(* CODESYS project PartX_Codesys

Project tree, tasks and I/O mapping:
  Device : CODESYS Control Win V3 x64, CODESYS, version 3.5.22.10
    application Application
      libraries: Standard, 3.5.22.0 (System); VisuDialogs, * (System); CAA Net Base Services, * (CAA Technical Workgroup)
      task ENIPScannerIOTask (cyclic, interval t#10ms, priority 0) calls EtherNet_IP_Scanner.IOCycle
      task ENIPScannerServiceTask (cyclic, interval t#20ms, priority 30) calls EtherNet_IP_Scanner.ServiceCycle
      task MainTask (cyclic, interval t#20ms, priority 1) calls F001_SR00_MAIN, F002_SR00_MAIN
      task VISU_TASK (cyclic, interval 100 ms, priority 31) calls VisuElems.Visu_Prg
      F001_ROBOT/
        program F001_SR00_MAIN [?]
        program F001_SR02_RBT_ERRORS [?]
        program F001_SR03_STEPS [?]
        program F001_SR04_RBT_INIT [?]
        program F001_SR05_SET_TRF [?]
        program F001_SR06_RBT_MOTIONS [?]
        program F001_SR07_CAMERA [?]
        program F001_SR08_Explicit [ST]
        program F001_SR08_Explicit_Messaging [ST]
        program F001_SR08_ExplicitMessaging [?]
        function block RobotHandshake [ST]
      F002_PART_X/
        program F002_SR00_MAIN [?]
        program F002_SR01_SOCKET_SERVER [ST]
        program F002_SR02_SOCKET_CLIENT [ST]
        program F002_SR03_PARTX [?]: BOUNCE, CLEAR, IDLE, IDLE_Trigger, Manual_ACT, MOVE_FWD, MOVE_MANUAL, MOVE_REV, SCHED, SCHED_ACT
      F020_HMI_Pages/
        visualisation F020_Camera_Robot
        visualisation F020_PartX_Screen
        visualisation Visualization
      F1000_FBs/
        Meca500/
          function block Delay [ST]
          function block GetErrors [ST]
          function block Gripper [ST]
          function block MoveGripper [ST]
          function block MoveJoints [ST]
          function block MoveJointsRel [ST]
          function block MoveJointsVel [ST]
          function block MoveLin [ST]
          function block MoveLinRelTrf [ST]
          function block MoveLinRelWrf [ST]
          function block MoveLinVelTrf [ST]
          function block MoveLinVelWrf [ST]
          function block MovePose [ST]
          function block SetAutoConf [ST]
          function block SetAutoConfTurn [ST]
          function block SetBlending [ST]
          function block SetCartAcc [ST]
          function block SetCartAngVel [ST]
          function block SetCartLinVel [ST]
          function block SetCheckpoint [ST]
          function block SetConf [ST]
          function block SetConfTurn [ST]
          function block SetGripperForce [ST]
          function block SetGripperRange [ST]
          function block SetGripperVel [ST]
          function block SetJointAcc [ST]
          function block SetJointsVelLimit [ST]
          function block SetJointVel [ST]
          function block SetTorqueLimitCfg [ST]
          function block SetTorqueLimits [ST]
          function block SetTrf [ST]
          function block SetValveState [ST]
          function block SetVelTimeout [ST]
          function block SetWrf [ST]
          function block StartProgram [ST]
          Utiliy/
            function block CalculateWRF [ST]
      F1000_UDTs/
        data type E_SchedState
        data type UDT_Explicit
        UDT_Meca500/
          ENUM/
            data type Meca500_DynamicDataTypeID
            data type Meca500_Errors
            data type Meca500_MotionCommandID
          STRUCT/
            data type Meca500
            Meca500_Inputs/
              data type Meca500_DynamicData
              data type Meca500_Inputs
              data type Meca500_Motion
              data type Meca500_MotionStatus
              data type Meca500_RobotStatus
              data type Meca500_Status
              data type Meca500_TimeStamp
            Meca500_Outputs/
              data type Meca500_BrakeControl
              data type Meca500_MotionCommand
              data type Meca500_MotionControl
              data type Meca500_Outputs
              data type Meca500_RobotControl
        data type UDT_PARTX
        data type UDT_Robot
        data type UDT_StepConfig
        data type UDT_SYS
        data type UDT_VS_Series
      F100_VARs/
        global variables GVL
        text list TL_Directions
      program PLC_PRG [ST]
    Ethernet : Ethernet, CODESYS, version 4.2.0.0
        settings: IPAddress = [192,168,0,247]; SubnetMask = [255,255,255,0]; GatewayAddress = [0,0,0,0]; MACAddress = [16#E8,16#97,16#44,16#1A,16#95,16#04]; NetworkInterfaceName = 'Ethernet'; NetworkInterfaceName = "Ethernet"; SaveCommunicationSettings = FALSE; IPAddress = [192,168,0,2]; SubnetMask = [255,255,255,0]; GatewayAddress = [0,0,0,0]
      EtherNet_IP_Scanner : EtherNet/IP Scanner, CODESYS, order no. 1, version 4.8.0.0
        FANUC_Robot : Generic EtherNet/IP device, CODESYS, version 4.6.0.0
            settings: INITIALIZED = TRUE; IP address of Target = [16#C0,16#A8,16#00,16#01]; Keying.Check Device Type = FALSE; Keying.Check Vendor Code = FALSE; Keying.Check Product Code = FALSE; Keying.Check Major Revision = FALSE; Keying.Check Minor Revision = FALSE; RequiredConfigVersion = 50660864; Number of Connections = 1; Connection Settings.Requested packet interval = 32000 µs; Connection Settings.OT Connection Parameters = 18502; Connection Settings.TO Connection Parameters = 18498; Connection Settings.Connection Flags = 1056; Connection Settings.Connection Path Size = 8; Connection Settings.Large OT Connection Parameters = 1207959622; Connection Settings.Large TO Connection Parameters = 1207959618; Connection Path = [16#20,16#04,16#24,16#64,16#2C,16#97,16#2C,16#65]; Heartbeat Multiplier = 1; Input_Param0.ReadOnly = False; Input_Param0.BitSize = 8; Input_Param0.DataSize = 1; Input_Param1.ReadOnly = False; Input_Param1.BitSize = 8; Input_Param1.DataSize = 1; Input_Param2.ReadOnly = False; Input_Param2.BitSize = 8; Input_Param2.DataSize = 1; Input_Param3.ReadOnly = False; Input_Param3.BitSize = 8; Input_Param3.DataSize = 1; Input_Param4.ReadOnly = False; Input_Param4.BitSize = 8; Input_Param4.DataSize = 1; Input_Param5.ReadOnly = False; Input_Param5.BitSize = 8; Input_Param5.DataSize = 1; Input_Param6.ReadOnly = False; Input_Param6.BitSize = 8; Input_Param6.DataSize = 1; Input_Param7.ReadOnly = False;
              Input_Param7.BitSize = 8; Input_Param7.DataSize = 1; Input_Param8.ReadOnly = False; Input_Param8.BitSize = 8; Input_Param8.DataSize = 1; Input_Param9.ReadOnly = False; Input_Param9.BitSize = 8; Input_Param9.DataSize = 1; Input_Param10.ReadOnly = False; Input_Param10.BitSize = 8; Input_Param10.DataSize = 1; Input_Param11.ReadOnly = False; Input_Param11.BitSize = 8; Input_Param11.DataSize = 1; Input_Param12.ReadOnly = False; Input_Param12.BitSize = 8; Input_Param12.DataSize = 1; Input_Param13.ReadOnly = False; Input_Param13.BitSize = 8; Input_Param13.DataSize = 1; Input_Param14.ReadOnly = False; Input_Param14.BitSize = 8; Input_Param14.DataSize = 1; Input_Param15.ReadOnly = False; Input_Param15.BitSize = 8; Input_Param15.DataSize = 1; Input_Param16.ReadOnly = False; Input_Param16.BitSize = 8; Input_Param16.DataSize = 1; Input_Param17.ReadOnly = False; Input_Param17.BitSize = 8; Input_Param17.DataSize = 1; Input_Param18.ReadOnly = False; Input_Param18.BitSize = 8; Input_Param18.DataSize = 1; Input_Param19.ReadOnly = False; Input_Param19.BitSize = 8; Input_Param19.DataSize = 1; Input_Param20.ReadOnly = False; Input_Param20.BitSize = 8;
              Input_Param20.DataSize = 1; Input_Param21.ReadOnly = False; Input_Param21.BitSize = 8; Input_Param21.DataSize = 1; Input_Param22.ReadOnly = False; Input_Param22.BitSize = 8; Input_Param22.DataSize = 1; Input_Param23.ReadOnly = False; Input_Param23.BitSize = 8; Input_Param23.DataSize = 1; Input_Param24.ReadOnly = False; Input_Param24.BitSize = 8; Input_Param24.DataSize = 1; Input_Param25.ReadOnly = False; Input_Param25.BitSize = 8; Input_Param25.DataSize = 1; Input_Param26.ReadOnly = False; Input_Param26.BitSize = 8; Input_Param26.DataSize = 1; Input_Param27.ReadOnly = False; Input_Param27.BitSize = 8; Input_Param27.DataSize = 1; Input_Param28.ReadOnly = False; Input_Param28.BitSize = 8; Input_Param28.DataSize = 1; Input_Param29.ReadOnly = False; Input_Param29.BitSize = 8; Input_Param29.DataSize = 1; Input_Param30.ReadOnly = False; Input_Param30.BitSize = 8; Input_Param30.DataSize = 1; Input_Param31.ReadOnly = False; Input_Param31.BitSize = 8; Input_Param31.DataSize = 1; Input_Param32.ReadOnly = False; Input_Param32.BitSize = 8; Input_Param32.DataSize = 1; Input_Param33.ReadOnly = False; Input_Param33.BitSize = 8; Input_Param33.DataSize = 1;
              Input_Param34.ReadOnly = False; Input_Param34.BitSize = 8; Input_Param34.DataSize = 1; Input_Param35.ReadOnly = False; Input_Param35.BitSize = 8; Input_Param35.DataSize = 1; Input_Param36.ReadOnly = False; Input_Param36.BitSize = 8; Input_Param36.DataSize = 1; Input_Param37.ReadOnly = False; Input_Param37.BitSize = 8; Input_Param37.DataSize = 1; Input_Param38.ReadOnly = False; Input_Param38.BitSize = 8; Input_Param38.DataSize = 1; Input_Param39.ReadOnly = False; Input_Param39.BitSize = 8; Input_Param39.DataSize = 1; Input_Param40.ReadOnly = False; Input_Param40.BitSize = 8; Input_Param40.DataSize = 1; Input_Param41.ReadOnly = False; Input_Param41.BitSize = 8; Input_Param41.DataSize = 1; Input_Param42.ReadOnly = False; Input_Param42.BitSize = 8; Input_Param42.DataSize = 1; Input_Param43.ReadOnly = False; Input_Param43.BitSize = 8; Input_Param43.DataSize = 1; Input_Param44.ReadOnly = False; Input_Param44.BitSize = 8; Input_Param44.DataSize = 1; Input_Param45.ReadOnly = False; Input_Param45.BitSize = 8; Input_Param45.DataSize = 1; Input_Param46.ReadOnly = False; Input_Param46.BitSize = 8; Input_Param46.DataSize = 1; Input_Param47.ReadOnly = False;
              Input_Param47.BitSize = 8; Input_Param47.DataSize = 1; Input_Param48.ReadOnly = False; Input_Param48.BitSize = 8; Input_Param48.DataSize = 1; Input_Param49.ReadOnly = False; Input_Param49.BitSize = 8; Input_Param49.DataSize = 1; Input_Param50.ReadOnly = False; Input_Param50.BitSize = 8; Input_Param50.DataSize = 1; Input_Param51.ReadOnly = False; Input_Param51.BitSize = 8; Input_Param51.DataSize = 1; Input_Param52.ReadOnly = False; Input_Param52.BitSize = 8; Input_Param52.DataSize = 1; Input_Param53.ReadOnly = False; Input_Param53.BitSize = 8; Input_Param53.DataSize = 1; Input_Param54.ReadOnly = False; Input_Param54.BitSize = 8; Input_Param54.DataSize = 1; Input_Param55.ReadOnly = False; Input_Param55.BitSize = 8; Input_Param55.DataSize = 1; Input_Param56.ReadOnly = False; Input_Param56.BitSize = 8; Input_Param56.DataSize = 1; Input_Param57.ReadOnly = False; Input_Param57.BitSize = 8; Input_Param57.DataSize = 1; Input_Param58.ReadOnly = False; Input_Param58.BitSize = 8; Input_Param58.DataSize = 1; Input_Param59.ReadOnly = False; Input_Param59.BitSize = 8; Input_Param59.DataSize = 1; Input_Param60.ReadOnly = False; Input_Param60.BitSize = 8;
              Input_Param60.DataSize = 1; Input_Param61.ReadOnly = False; Input_Param61.BitSize = 8; Input_Param61.DataSize = 1; Input_Param62.ReadOnly = False; Input_Param62.BitSize = 8; Input_Param62.DataSize = 1; Input_Param63.ReadOnly = False; Input_Param63.BitSize = 8; Input_Param63.DataSize = 1; Output_Param0.ReadOnly = False; Output_Param0.BitSize = 8; Output_Param0.DataSize = 1; Output_Param1.ReadOnly = False; Output_Param1.BitSize = 8; Output_Param1.DataSize = 1; Output_Param2.ReadOnly = False; Output_Param2.BitSize = 8; Output_Param2.DataSize = 1; Output_Param3.ReadOnly = False; Output_Param3.BitSize = 8; Output_Param3.DataSize = 1; Output_Param4.ReadOnly = False; Output_Param4.BitSize = 8; Output_Param4.DataSize = 1; Output_Param5.ReadOnly = False; Output_Param5.BitSize = 8; Output_Param5.DataSize = 1; Output_Param6.ReadOnly = False; Output_Param6.BitSize = 8; Output_Param6.DataSize = 1; Output_Param7.ReadOnly = False; Output_Param7.BitSize = 8; Output_Param7.DataSize = 1; Output_Param8.ReadOnly = False; Output_Param8.BitSize = 8; Output_Param8.DataSize = 1; Output_Param9.ReadOnly = False; Output_Param9.BitSize = 8; Output_Param9.DataSize = 1;
              Output_Param10.ReadOnly = False; Output_Param10.BitSize = 8; Output_Param10.DataSize = 1; Output_Param11.ReadOnly = False; Output_Param11.BitSize = 8; Output_Param11.DataSize = 1; Output_Param12.ReadOnly = False; Output_Param12.BitSize = 8; Output_Param12.DataSize = 1; Output_Param13.ReadOnly = False; Output_Param13.BitSize = 8; Output_Param13.DataSize = 1; Output_Param14.ReadOnly = False; Output_Param14.BitSize = 8; Output_Param14.DataSize = 1; Output_Param15.ReadOnly = False; Output_Param15.BitSize = 8; Output_Param15.DataSize = 1; Output_Param16.ReadOnly = False; Output_Param16.BitSize = 8; Output_Param16.DataSize = 1; Output_Param17.ReadOnly = False; Output_Param17.BitSize = 8; Output_Param17.DataSize = 1; Output_Param18.ReadOnly = False; Output_Param18.BitSize = 8; Output_Param18.DataSize = 1; Output_Param19.ReadOnly = False; Output_Param19.BitSize = 8; Output_Param19.DataSize = 1; Output_Param20.ReadOnly = False; Output_Param20.BitSize = 8; Output_Param20.DataSize = 1; Output_Param21.ReadOnly = False; Output_Param21.BitSize = 8; Output_Param21.DataSize = 1; Output_Param22.ReadOnly = False; Output_Param22.BitSize = 8; Output_Param22.DataSize = 1; Output_Param23.ReadOnly = False;
              Output_Param23.BitSize = 8; Output_Param23.DataSize = 1; Output_Param24.ReadOnly = False; Output_Param24.BitSize = 8; Output_Param24.DataSize = 1; Output_Param25.ReadOnly = False; Output_Param25.BitSize = 8; Output_Param25.DataSize = 1; Output_Param26.ReadOnly = False; Output_Param26.BitSize = 8; Output_Param26.DataSize = 1; Output_Param27.ReadOnly = False; Output_Param27.BitSize = 8; Output_Param27.DataSize = 1; Output_Param28.ReadOnly = False; Output_Param28.BitSize = 8; Output_Param28.DataSize = 1; Output_Param29.ReadOnly = False; Output_Param29.BitSize = 8; Output_Param29.DataSize = 1; Output_Param30.ReadOnly = False; Output_Param30.BitSize = 8; Output_Param30.DataSize = 1; Output_Param31.ReadOnly = False; Output_Param31.BitSize = 8; Output_Param31.DataSize = 1; Output_Param32.ReadOnly = False; Output_Param32.BitSize = 8; Output_Param32.DataSize = 1; Output_Param33.ReadOnly = False; Output_Param33.BitSize = 8; Output_Param33.DataSize = 1; Output_Param34.ReadOnly = False; Output_Param34.BitSize = 8; Output_Param34.DataSize = 1; Output_Param35.ReadOnly = False; Output_Param35.BitSize = 8; Output_Param35.DataSize = 1; Output_Param36.ReadOnly = False; Output_Param36.BitSize = 8;
              Output_Param36.DataSize = 1; Output_Param37.ReadOnly = False; Output_Param37.BitSize = 8; Output_Param37.DataSize = 1; Output_Param38.ReadOnly = False; Output_Param38.BitSize = 8; Output_Param38.DataSize = 1; Output_Param39.ReadOnly = False; Output_Param39.BitSize = 8; Output_Param39.DataSize = 1; Output_Param40.ReadOnly = False; Output_Param40.BitSize = 8; Output_Param40.DataSize = 1; Output_Param41.ReadOnly = False; Output_Param41.BitSize = 8; Output_Param41.DataSize = 1; Output_Param42.ReadOnly = False; Output_Param42.BitSize = 8; Output_Param42.DataSize = 1; Output_Param43.ReadOnly = False; Output_Param43.BitSize = 8; Output_Param43.DataSize = 1; Output_Param44.ReadOnly = False; Output_Param44.BitSize = 8; Output_Param44.DataSize = 1; Output_Param45.ReadOnly = False; Output_Param45.BitSize = 8; Output_Param45.DataSize = 1; Output_Param46.ReadOnly = False; Output_Param46.BitSize = 8; Output_Param46.DataSize = 1; Output_Param47.ReadOnly = False; Output_Param47.BitSize = 8; Output_Param47.DataSize = 1; Output_Param48.ReadOnly = False; Output_Param48.BitSize = 8; Output_Param48.DataSize = 1; Output_Param49.ReadOnly = False; Output_Param49.BitSize = 8; Output_Param49.DataSize = 1;
              Output_Param50.ReadOnly = False; Output_Param50.BitSize = 8; Output_Param50.DataSize = 1; Output_Param51.ReadOnly = False; Output_Param51.BitSize = 8; Output_Param51.DataSize = 1; Output_Param52.ReadOnly = False; Output_Param52.BitSize = 8; Output_Param52.DataSize = 1; Output_Param53.ReadOnly = False; Output_Param53.BitSize = 8; Output_Param53.DataSize = 1; Output_Param54.ReadOnly = False; Output_Param54.BitSize = 8; Output_Param54.DataSize = 1; Output_Param55.ReadOnly = False; Output_Param55.BitSize = 8; Output_Param55.DataSize = 1; Output_Param56.ReadOnly = False; Output_Param56.BitSize = 8; Output_Param56.DataSize = 1; Output_Param57.ReadOnly = False; Output_Param57.BitSize = 8; Output_Param57.DataSize = 1; Output_Param58.ReadOnly = False; Output_Param58.BitSize = 8; Output_Param58.DataSize = 1; Output_Param59.ReadOnly = False; Output_Param59.BitSize = 8; Output_Param59.DataSize = 1; Output_Param60.ReadOnly = False; Output_Param60.BitSize = 8; Output_Param60.DataSize = 1; Output_Param61.ReadOnly = False; Output_Param61.BitSize = 8; Output_Param61.DataSize = 1; Output_Param62.ReadOnly = False; Output_Param62.BitSize = 8; Output_Param62.DataSize = 1; Output_Param63.ReadOnly = False;
              Output_Param63.BitSize = 8; Output_Param63.DataSize = 1; Input_Param0.Name = 'Input_Param0'; Input_Param0.HelpString = ''; Input_Param0.ReadOnly = False; Input_Param0.BitSize = 8; Input_Param0.DataSize = 1; Input_Param0.DataType = 'BYTE'; Input_Param1.Name = 'Input_Param1'; Input_Param1.HelpString = ''; Input_Param1.ReadOnly = False; Input_Param1.BitSize = 8; Input_Param1.DataSize = 1; Input_Param1.DataType = 'BYTE'; Input_Param2.Name = 'Input_Param2'; Input_Param2.HelpString = ''; Input_Param2.ReadOnly = False; Input_Param2.BitSize = 8; Input_Param2.DataSize = 1; Input_Param2.DataType = 'BYTE'; Input_Param3.Name = 'Input_Param3'; Input_Param3.HelpString = ''; Input_Param3.ReadOnly = False; Input_Param3.BitSize = 8; Input_Param3.DataSize = 1; Input_Param3.DataType = 'BYTE'; Input_Param4.Name = 'Input_Param4'; Input_Param4.HelpString = ''; Input_Param4.ReadOnly = False; Input_Param4.BitSize = 8; Input_Param4.DataSize = 1; Input_Param4.DataType = 'BYTE'; Input_Param5.Name = 'Input_Param5'; Input_Param5.HelpString = ''; Input_Param5.ReadOnly = False; Input_Param5.BitSize = 8; Input_Param5.DataSize = 1; Input_Param5.DataType = 'BYTE'; Input_Param6.Name = 'Input_Param6'; Input_Param6.HelpString = '';
              Input_Param6.ReadOnly = False; Input_Param6.BitSize = 8; Input_Param6.DataSize = 1; Input_Param6.DataType = 'BYTE'; Input_Param7.Name = 'Input_Param7'; Input_Param7.HelpString = ''; Input_Param7.ReadOnly = False; Input_Param7.BitSize = 8; Input_Param7.DataSize = 1; Input_Param7.DataType = 'BYTE'; Input_Param8.Name = 'Input_Param8'; Input_Param8.HelpString = ''; Input_Param8.ReadOnly = False; Input_Param8.BitSize = 8; Input_Param8.DataSize = 1; Input_Param8.DataType = 'BYTE'; Input_Param9.Name = 'Input_Param9'; Input_Param9.HelpString = ''; Input_Param9.ReadOnly = False; Input_Param9.BitSize = 8; Input_Param9.DataSize = 1; Input_Param9.DataType = 'BYTE'; Input_Param10.Name = 'Input_Param10'; Input_Param10.HelpString = ''; Input_Param10.ReadOnly = False; Input_Param10.BitSize = 8; Input_Param10.DataSize = 1; Input_Param10.DataType = 'BYTE'; Input_Param11.Name = 'Input_Param11'; Input_Param11.HelpString = ''; Input_Param11.ReadOnly = False; Input_Param11.BitSize = 8; Input_Param11.DataSize = 1; Input_Param11.DataType = 'BYTE'; Input_Param12.Name = 'Input_Param12'; Input_Param12.HelpString = ''; Input_Param12.ReadOnly = False; Input_Param12.BitSize = 8; Input_Param12.DataSize = 1; Input_Param12.DataType = 'BYTE';
              Input_Param13.Name = 'Input_Param13'; Input_Param13.HelpString = ''; Input_Param13.ReadOnly = False; Input_Param13.BitSize = 8; Input_Param13.DataSize = 1; Input_Param13.DataType = 'BYTE'; Input_Param14.Name = 'Input_Param14'; Input_Param14.HelpString = ''; Input_Param14.ReadOnly = False; Input_Param14.BitSize = 8; Input_Param14.DataSize = 1; Input_Param14.DataType = 'BYTE'; Input_Param15.Name = 'Input_Param15'; Input_Param15.HelpString = ''; Input_Param15.ReadOnly = False; Input_Param15.BitSize = 8; Input_Param15.DataSize = 1; Input_Param15.DataType = 'BYTE'; Input_Param16.Name = 'Input_Param16'; Input_Param16.HelpString = ''; Input_Param16.ReadOnly = False; Input_Param16.BitSize = 8; Input_Param16.DataSize = 1; Input_Param16.DataType = 'BYTE'; Input_Param17.Name = 'Input_Param17'; Input_Param17.HelpString = ''; Input_Param17.ReadOnly = False; Input_Param17.BitSize = 8; Input_Param17.DataSize = 1; Input_Param17.DataType = 'BYTE'; Input_Param18.Name = 'Input_Param18'; Input_Param18.HelpString = ''; Input_Param18.ReadOnly = False; Input_Param18.BitSize = 8; Input_Param18.DataSize = 1; Input_Param18.DataType = 'BYTE'; Input_Param19.Name = 'Input_Param19'; Input_Param19.HelpString = ''; Input_Param19.ReadOnly = False; Input_Param19.BitSize = 8;
              Input_Param19.DataSize = 1; Input_Param19.DataType = 'BYTE'; Input_Param20.Name = 'Input_Param20'; Input_Param20.HelpString = ''; Input_Param20.ReadOnly = False; Input_Param20.BitSize = 8; Input_Param20.DataSize = 1; Input_Param20.DataType = 'BYTE'; Input_Param21.Name = 'Input_Param21'; Input_Param21.HelpString = ''; Input_Param21.ReadOnly = False; Input_Param21.BitSize = 8; Input_Param21.DataSize = 1; Input_Param21.DataType = 'BYTE'; Input_Param22.Name = 'Input_Param22'; Input_Param22.HelpString = ''; Input_Param22.ReadOnly = False; Input_Param22.BitSize = 8; Input_Param22.DataSize = 1; Input_Param22.DataType = 'BYTE'; Input_Param23.Name = 'Input_Param23'; Input_Param23.HelpString = ''; Input_Param23.ReadOnly = False; Input_Param23.BitSize = 8; Input_Param23.DataSize = 1; Input_Param23.DataType = 'BYTE'; Input_Param24.Name = 'Input_Param24'; Input_Param24.HelpString = ''; Input_Param24.ReadOnly = False; Input_Param24.BitSize = 8; Input_Param24.DataSize = 1; Input_Param24.DataType = 'BYTE'; Input_Param25.Name = 'Input_Param25'; Input_Param25.HelpString = ''; Input_Param25.ReadOnly = False; Input_Param25.BitSize = 8; Input_Param25.DataSize = 1; Input_Param25.DataType = 'BYTE'; Input_Param26.Name = 'Input_Param26'; Input_Param26.HelpString = '';
              Input_Param26.ReadOnly = False; Input_Param26.BitSize = 8; Input_Param26.DataSize = 1; Input_Param26.DataType = 'BYTE'; Input_Param27.Name = 'Input_Param27'; Input_Param27.HelpString = ''; Input_Param27.ReadOnly = False; Input_Param27.BitSize = 8; Input_Param27.DataSize = 1; Input_Param27.DataType = 'BYTE'; Input_Param28.Name = 'Input_Param28'; Input_Param28.HelpString = ''; Input_Param28.ReadOnly = False; Input_Param28.BitSize = 8; Input_Param28.DataSize = 1; Input_Param28.DataType = 'BYTE'; Input_Param29.Name = 'Input_Param29'; Input_Param29.HelpString = ''; Input_Param29.ReadOnly = False; Input_Param29.BitSize = 8; Input_Param29.DataSize = 1; Input_Param29.DataType = 'BYTE'; Input_Param30.Name = 'Input_Param30'; Input_Param30.HelpString = ''; Input_Param30.ReadOnly = False; Input_Param30.BitSize = 8; Input_Param30.DataSize = 1; Input_Param30.DataType = 'BYTE'; Input_Param31.Name = 'Input_Param31'; Input_Param31.HelpString = ''; Input_Param31.ReadOnly = False; Input_Param31.BitSize = 8; Input_Param31.DataSize = 1; Input_Param31.DataType = 'BYTE'; Input_Param32.Name = 'Input_Param32'; Input_Param32.HelpString = ''; Input_Param32.ReadOnly = False; Input_Param32.BitSize = 8; Input_Param32.DataSize = 1; Input_Param32.DataType = 'BYTE';
              Input_Param33.Name = 'Input_Param33'; Input_Param33.HelpString = ''; Input_Param33.ReadOnly = False; Input_Param33.BitSize = 8; Input_Param33.DataSize = 1; Input_Param33.DataType = 'BYTE'; Input_Param34.Name = 'Input_Param34'; Input_Param34.HelpString = ''; Input_Param34.ReadOnly = False; Input_Param34.BitSize = 8; Input_Param34.DataSize = 1; Input_Param34.DataType = 'BYTE'; Input_Param35.Name = 'Input_Param35'; Input_Param35.HelpString = ''; Input_Param35.ReadOnly = False; Input_Param35.BitSize = 8; Input_Param35.DataSize = 1; Input_Param35.DataType = 'BYTE'; Input_Param36.Name = 'Input_Param36'; Input_Param36.HelpString = ''; Input_Param36.ReadOnly = False; Input_Param36.BitSize = 8; Input_Param36.DataSize = 1; Input_Param36.DataType = 'BYTE'; Input_Param37.Name = 'Input_Param37'; Input_Param37.HelpString = ''; Input_Param37.ReadOnly = False; Input_Param37.BitSize = 8; Input_Param37.DataSize = 1; Input_Param37.DataType = 'BYTE'; Input_Param38.Name = 'Input_Param38'; Input_Param38.HelpString = ''; Input_Param38.ReadOnly = False; Input_Param38.BitSize = 8; Input_Param38.DataSize = 1; Input_Param38.DataType = 'BYTE'; Input_Param39.Name = 'Input_Param39'; Input_Param39.HelpString = ''; Input_Param39.ReadOnly = False; Input_Param39.BitSize = 8;
              Input_Param39.DataSize = 1; Input_Param39.DataType = 'BYTE'; Input_Param40.Name = 'Input_Param40'; Input_Param40.HelpString = ''; Input_Param40.ReadOnly = False; Input_Param40.BitSize = 8; Input_Param40.DataSize = 1; Input_Param40.DataType = 'BYTE'; Input_Param41.Name = 'Input_Param41'; Input_Param41.HelpString = ''; Input_Param41.ReadOnly = False; Input_Param41.BitSize = 8; Input_Param41.DataSize = 1; Input_Param41.DataType = 'BYTE'; Input_Param42.Name = 'Input_Param42'; Input_Param42.HelpString = ''; Input_Param42.ReadOnly = False; Input_Param42.BitSize = 8; Input_Param42.DataSize = 1; Input_Param42.DataType = 'BYTE'; Input_Param43.Name = 'Input_Param43'; Input_Param43.HelpString = ''; Input_Param43.ReadOnly = False; Input_Param43.BitSize = 8; Input_Param43.DataSize = 1; Input_Param43.DataType = 'BYTE'; Input_Param44.Name = 'Input_Param44'; Input_Param44.HelpString = ''; Input_Param44.ReadOnly = False; Input_Param44.BitSize = 8; Input_Param44.DataSize = 1; Input_Param44.DataType = 'BYTE'; Input_Param45.Name = 'Input_Param45'; Input_Param45.HelpString = ''; Input_Param45.ReadOnly = False; Input_Param45.BitSize = 8; Input_Param45.DataSize = 1; Input_Param45.DataType = 'BYTE'; Input_Param46.Name = 'Input_Param46'; Input_Param46.HelpString = '';
              Input_Param46.ReadOnly = False; Input_Param46.BitSize = 8; Input_Param46.DataSize = 1; Input_Param46.DataType = 'BYTE'; Input_Param47.Name = 'Input_Param47'; Input_Param47.HelpString = ''; Input_Param47.ReadOnly = False; Input_Param47.BitSize = 8; Input_Param47.DataSize = 1; Input_Param47.DataType = 'BYTE'; Input_Param48.Name = 'Input_Param48'; Input_Param48.HelpString = ''; Input_Param48.ReadOnly = False; Input_Param48.BitSize = 8; Input_Param48.DataSize = 1; Input_Param48.DataType = 'BYTE'; Input_Param49.Name = 'Input_Param49'; Input_Param49.HelpString = ''; Input_Param49.ReadOnly = False; Input_Param49.BitSize = 8; Input_Param49.DataSize = 1; Input_Param49.DataType = 'BYTE'; Input_Param50.Name = 'Input_Param50'; Input_Param50.HelpString = ''; Input_Param50.ReadOnly = False; Input_Param50.BitSize = 8; Input_Param50.DataSize = 1; Input_Param50.DataType = 'BYTE'; Input_Param51.Name = 'Input_Param51'; Input_Param51.HelpString = ''; Input_Param51.ReadOnly = False; Input_Param51.BitSize = 8; Input_Param51.DataSize = 1; Input_Param51.DataType = 'BYTE'; Input_Param52.Name = 'Input_Param52'; Input_Param52.HelpString = ''; Input_Param52.ReadOnly = False; Input_Param52.BitSize = 8; Input_Param52.DataSize = 1; Input_Param52.DataType = 'BYTE';
              Input_Param53.Name = 'Input_Param53'; Input_Param53.HelpString = ''; Input_Param53.ReadOnly = False; Input_Param53.BitSize = 8; Input_Param53.DataSize = 1; Input_Param53.DataType = 'BYTE'; Input_Param54.Name = 'Input_Param54'; Input_Param54.HelpString = ''; Input_Param54.ReadOnly = False; Input_Param54.BitSize = 8; Input_Param54.DataSize = 1; Input_Param54.DataType = 'BYTE'; Input_Param55.Name = 'Input_Param55'; Input_Param55.HelpString = ''; Input_Param55.ReadOnly = False; Input_Param55.BitSize = 8; Input_Param55.DataSize = 1; Input_Param55.DataType = 'BYTE'; Input_Param56.Name = 'Input_Param56'; Input_Param56.HelpString = ''; Input_Param56.ReadOnly = False; Input_Param56.BitSize = 8; Input_Param56.DataSize = 1; Input_Param56.DataType = 'BYTE'; Input_Param57.Name = 'Input_Param57'; Input_Param57.HelpString = ''; Input_Param57.ReadOnly = False; Input_Param57.BitSize = 8; Input_Param57.DataSize = 1; Input_Param57.DataType = 'BYTE'; Input_Param58.Name = 'Input_Param58'; Input_Param58.HelpString = ''; Input_Param58.ReadOnly = False; Input_Param58.BitSize = 8; Input_Param58.DataSize = 1; Input_Param58.DataType = 'BYTE'; Input_Param59.Name = 'Input_Param59'; Input_Param59.HelpString = ''; Input_Param59.ReadOnly = False; Input_Param59.BitSize = 8;
              Input_Param59.DataSize = 1; Input_Param59.DataType = 'BYTE'; Input_Param60.Name = 'Input_Param60'; Input_Param60.HelpString = ''; Input_Param60.ReadOnly = False; Input_Param60.BitSize = 8; Input_Param60.DataSize = 1; Input_Param60.DataType = 'BYTE'; Input_Param61.Name = 'Input_Param61'; Input_Param61.HelpString = ''; Input_Param61.ReadOnly = False; Input_Param61.BitSize = 8; Input_Param61.DataSize = 1; Input_Param61.DataType = 'BYTE'; Input_Param62.Name = 'Input_Param62'; Input_Param62.HelpString = ''; Input_Param62.ReadOnly = False; Input_Param62.BitSize = 8; Input_Param62.DataSize = 1; Input_Param62.DataType = 'BYTE'; Input_Param63.Name = 'Input_Param63'; Input_Param63.HelpString = ''; Input_Param63.ReadOnly = False; Input_Param63.BitSize = 8; Input_Param63.DataSize = 1; Input_Param63.DataType = 'BYTE'; Output_Param0.Name = 'Output_Param0'; Output_Param0.HelpString = ''; Output_Param0.ReadOnly = False; Output_Param0.BitSize = 8; Output_Param0.DataSize = 1; Output_Param0.DataType = 'BYTE'; Output_Param1.Name = 'Output_Param1'; Output_Param1.HelpString = ''; Output_Param1.ReadOnly = False; Output_Param1.BitSize = 8; Output_Param1.DataSize = 1; Output_Param1.DataType = 'BYTE'; Output_Param2.Name = 'Output_Param2'; Output_Param2.HelpString = '';
              Output_Param2.ReadOnly = False; Output_Param2.BitSize = 8; Output_Param2.DataSize = 1; Output_Param2.DataType = 'BYTE'; Output_Param3.Name = 'Output_Param3'; Output_Param3.HelpString = ''; Output_Param3.ReadOnly = False; Output_Param3.BitSize = 8; Output_Param3.DataSize = 1; Output_Param3.DataType = 'BYTE'; Output_Param4.Name = 'Output_Param4'; Output_Param4.HelpString = ''; Output_Param4.ReadOnly = False; Output_Param4.BitSize = 8; Output_Param4.DataSize = 1; Output_Param4.DataType = 'BYTE'; Output_Param5.Name = 'Output_Param5'; Output_Param5.HelpString = ''; Output_Param5.ReadOnly = False; Output_Param5.BitSize = 8; Output_Param5.DataSize = 1; Output_Param5.DataType = 'BYTE'; Output_Param6.Name = 'Output_Param6'; Output_Param6.HelpString = ''; Output_Param6.ReadOnly = False; Output_Param6.BitSize = 8; Output_Param6.DataSize = 1; Output_Param6.DataType = 'BYTE'; Output_Param7.Name = 'Output_Param7'; Output_Param7.HelpString = ''; Output_Param7.ReadOnly = False; Output_Param7.BitSize = 8; Output_Param7.DataSize = 1; Output_Param7.DataType = 'BYTE'; Output_Param8.Name = 'Output_Param8'; Output_Param8.HelpString = ''; Output_Param8.ReadOnly = False; Output_Param8.BitSize = 8; Output_Param8.DataSize = 1; Output_Param8.DataType = 'BYTE';
              Output_Param9.Name = 'Output_Param9'; Output_Param9.HelpString = ''; Output_Param9.ReadOnly = False; Output_Param9.BitSize = 8; Output_Param9.DataSize = 1; Output_Param9.DataType = 'BYTE'; Output_Param10.Name = 'Output_Param10'; Output_Param10.HelpString = ''; Output_Param10.ReadOnly = False; Output_Param10.BitSize = 8; Output_Param10.DataSize = 1; Output_Param10.DataType = 'BYTE'; Output_Param11.Name = 'Output_Param11'; Output_Param11.HelpString = ''; Output_Param11.ReadOnly = False; Output_Param11.BitSize = 8; Output_Param11.DataSize = 1; Output_Param11.DataType = 'BYTE'; Output_Param12.Name = 'Output_Param12'; Output_Param12.HelpString = ''; Output_Param12.ReadOnly = False; Output_Param12.BitSize = 8; Output_Param12.DataSize = 1; Output_Param12.DataType = 'BYTE'; Output_Param13.Name = 'Output_Param13'; Output_Param13.HelpString = ''; Output_Param13.ReadOnly = False; Output_Param13.BitSize = 8; Output_Param13.DataSize = 1; Output_Param13.DataType = 'BYTE'; Output_Param14.Name = 'Output_Param14'; Output_Param14.HelpString = ''; Output_Param14.ReadOnly = False; Output_Param14.BitSize = 8; Output_Param14.DataSize = 1; Output_Param14.DataType = 'BYTE'; Output_Param15.Name = 'Output_Param15'; Output_Param15.HelpString = ''; Output_Param15.ReadOnly = False; Output_Param15.BitSize = 8;
              Output_Param15.DataSize = 1; Output_Param15.DataType = 'BYTE'; Output_Param16.Name = 'Output_Param16'; Output_Param16.HelpString = ''; Output_Param16.ReadOnly = False; Output_Param16.BitSize = 8; Output_Param16.DataSize = 1; Output_Param16.DataType = 'BYTE'; Output_Param17.Name = 'Output_Param17'; Output_Param17.HelpString = ''; Output_Param17.ReadOnly = False; Output_Param17.BitSize = 8; Output_Param17.DataSize = 1; Output_Param17.DataType = 'BYTE'; Output_Param18.Name = 'Output_Param18'; Output_Param18.HelpString = ''; Output_Param18.ReadOnly = False; Output_Param18.BitSize = 8; Output_Param18.DataSize = 1; Output_Param18.DataType = 'BYTE'; Output_Param19.Name = 'Output_Param19'; Output_Param19.HelpString = ''; Output_Param19.ReadOnly = False; Output_Param19.BitSize = 8; Output_Param19.DataSize = 1; Output_Param19.DataType = 'BYTE'; Output_Param20.Name = 'Output_Param20'; Output_Param20.HelpString = ''; Output_Param20.ReadOnly = False; Output_Param20.BitSize = 8; Output_Param20.DataSize = 1; Output_Param20.DataType = 'BYTE'; Output_Param21.Name = 'Output_Param21'; Output_Param21.HelpString = ''; Output_Param21.ReadOnly = False; Output_Param21.BitSize = 8; Output_Param21.DataSize = 1; Output_Param21.DataType = 'BYTE'; Output_Param22.Name = 'Output_Param22'; Output_Param22.HelpString = '';
              Output_Param22.ReadOnly = False; Output_Param22.BitSize = 8; Output_Param22.DataSize = 1; Output_Param22.DataType = 'BYTE'; Output_Param23.Name = 'Output_Param23'; Output_Param23.HelpString = ''; Output_Param23.ReadOnly = False; Output_Param23.BitSize = 8; Output_Param23.DataSize = 1; Output_Param23.DataType = 'BYTE'; Output_Param24.Name = 'Output_Param24'; Output_Param24.HelpString = ''; Output_Param24.ReadOnly = False; Output_Param24.BitSize = 8; Output_Param24.DataSize = 1; Output_Param24.DataType = 'BYTE'; Output_Param25.Name = 'Output_Param25'; Output_Param25.HelpString = ''; Output_Param25.ReadOnly = False; Output_Param25.BitSize = 8; Output_Param25.DataSize = 1; Output_Param25.DataType = 'BYTE'; Output_Param26.Name = 'Output_Param26'; Output_Param26.HelpString = ''; Output_Param26.ReadOnly = False; Output_Param26.BitSize = 8; Output_Param26.DataSize = 1; Output_Param26.DataType = 'BYTE'; Output_Param27.Name = 'Output_Param27'; Output_Param27.HelpString = ''; Output_Param27.ReadOnly = False; Output_Param27.BitSize = 8; Output_Param27.DataSize = 1; Output_Param27.DataType = 'BYTE'; Output_Param28.Name = 'Output_Param28'; Output_Param28.HelpString = ''; Output_Param28.ReadOnly = False; Output_Param28.BitSize = 8; Output_Param28.DataSize = 1; Output_Param28.DataType = 'BYTE';
              Output_Param29.Name = 'Output_Param29'; Output_Param29.HelpString = ''; Output_Param29.ReadOnly = False; Output_Param29.BitSize = 8; Output_Param29.DataSize = 1; Output_Param29.DataType = 'BYTE'; Output_Param30.Name = 'Output_Param30'; Output_Param30.HelpString = ''; Output_Param30.ReadOnly = False; Output_Param30.BitSize = 8; Output_Param30.DataSize = 1; Output_Param30.DataType = 'BYTE'; Output_Param31.Name = 'Output_Param31'; Output_Param31.HelpString = ''; Output_Param31.ReadOnly = False; Output_Param31.BitSize = 8; Output_Param31.DataSize = 1; Output_Param31.DataType = 'BYTE'; Output_Param32.Name = 'Output_Param32'; Output_Param32.HelpString = ''; Output_Param32.ReadOnly = False; Output_Param32.BitSize = 8; Output_Param32.DataSize = 1; Output_Param32.DataType = 'BYTE'; Output_Param33.Name = 'Output_Param33'; Output_Param33.HelpString = ''; Output_Param33.ReadOnly = False; Output_Param33.BitSize = 8; Output_Param33.DataSize = 1; Output_Param33.DataType = 'BYTE'; Output_Param34.Name = 'Output_Param34'; Output_Param34.HelpString = ''; Output_Param34.ReadOnly = False; Output_Param34.BitSize = 8; Output_Param34.DataSize = 1; Output_Param34.DataType = 'BYTE'; Output_Param35.Name = 'Output_Param35'; Output_Param35.HelpString = ''; Output_Param35.ReadOnly = False; Output_Param35.BitSize = 8;
              Output_Param35.DataSize = 1; Output_Param35.DataType = 'BYTE'; Output_Param36.Name = 'Output_Param36'; Output_Param36.HelpString = ''; Output_Param36.ReadOnly = False; Output_Param36.BitSize = 8; Output_Param36.DataSize = 1; Output_Param36.DataType = 'BYTE'; Output_Param37.Name = 'Output_Param37'; Output_Param37.HelpString = ''; Output_Param37.ReadOnly = False; Output_Param37.BitSize = 8; Output_Param37.DataSize = 1; Output_Param37.DataType = 'BYTE'; Output_Param38.Name = 'Output_Param38'; Output_Param38.HelpString = ''; Output_Param38.ReadOnly = False; Output_Param38.BitSize = 8; Output_Param38.DataSize = 1; Output_Param38.DataType = 'BYTE'; Output_Param39.Name = 'Output_Param39'; Output_Param39.HelpString = ''; Output_Param39.ReadOnly = False; Output_Param39.BitSize = 8; Output_Param39.DataSize = 1; Output_Param39.DataType = 'BYTE'; Output_Param40.Name = 'Output_Param40'; Output_Param40.HelpString = ''; Output_Param40.ReadOnly = False; Output_Param40.BitSize = 8; Output_Param40.DataSize = 1; Output_Param40.DataType = 'BYTE'; Output_Param41.Name = 'Output_Param41'; Output_Param41.HelpString = ''; Output_Param41.ReadOnly = False; Output_Param41.BitSize = 8; Output_Param41.DataSize = 1; Output_Param41.DataType = 'BYTE'; Output_Param42.Name = 'Output_Param42'; Output_Param42.HelpString = '';
              Output_Param42.ReadOnly = False; Output_Param42.BitSize = 8; Output_Param42.DataSize = 1; Output_Param42.DataType = 'BYTE'; Output_Param43.Name = 'Output_Param43'; Output_Param43.HelpString = ''; Output_Param43.ReadOnly = False; Output_Param43.BitSize = 8; Output_Param43.DataSize = 1; Output_Param43.DataType = 'BYTE'; Output_Param44.Name = 'Output_Param44'; Output_Param44.HelpString = ''; Output_Param44.ReadOnly = False; Output_Param44.BitSize = 8; Output_Param44.DataSize = 1; Output_Param44.DataType = 'BYTE'; Output_Param45.Name = 'Output_Param45'; Output_Param45.HelpString = ''; Output_Param45.ReadOnly = False; Output_Param45.BitSize = 8; Output_Param45.DataSize = 1; Output_Param45.DataType = 'BYTE'; Output_Param46.Name = 'Output_Param46'; Output_Param46.HelpString = ''; Output_Param46.ReadOnly = False; Output_Param46.BitSize = 8; Output_Param46.DataSize = 1; Output_Param46.DataType = 'BYTE'; Output_Param47.Name = 'Output_Param47'; Output_Param47.HelpString = ''; Output_Param47.ReadOnly = False; Output_Param47.BitSize = 8; Output_Param47.DataSize = 1; Output_Param47.DataType = 'BYTE'; Output_Param48.Name = 'Output_Param48'; Output_Param48.HelpString = ''; Output_Param48.ReadOnly = False; Output_Param48.BitSize = 8; Output_Param48.DataSize = 1; Output_Param48.DataType = 'BYTE';
              Output_Param49.Name = 'Output_Param49'; Output_Param49.HelpString = ''; Output_Param49.ReadOnly = False; Output_Param49.BitSize = 8; Output_Param49.DataSize = 1; Output_Param49.DataType = 'BYTE'; Output_Param50.Name = 'Output_Param50'; Output_Param50.HelpString = ''; Output_Param50.ReadOnly = False; Output_Param50.BitSize = 8; Output_Param50.DataSize = 1; Output_Param50.DataType = 'BYTE'; Output_Param51.Name = 'Output_Param51'; Output_Param51.HelpString = ''; Output_Param51.ReadOnly = False; Output_Param51.BitSize = 8; Output_Param51.DataSize = 1; Output_Param51.DataType = 'BYTE'; Output_Param52.Name = 'Output_Param52'; Output_Param52.HelpString = ''; Output_Param52.ReadOnly = False; Output_Param52.BitSize = 8; Output_Param52.DataSize = 1; Output_Param52.DataType = 'BYTE'; Output_Param53.Name = 'Output_Param53'; Output_Param53.HelpString = ''; Output_Param53.ReadOnly = False; Output_Param53.BitSize = 8; Output_Param53.DataSize = 1; Output_Param53.DataType = 'BYTE'; Output_Param54.Name = 'Output_Param54'; Output_Param54.HelpString = ''; Output_Param54.ReadOnly = False; Output_Param54.BitSize = 8; Output_Param54.DataSize = 1; Output_Param54.DataType = 'BYTE'; Output_Param55.Name = 'Output_Param55'; Output_Param55.HelpString = ''; Output_Param55.ReadOnly = False; Output_Param55.BitSize = 8;
              Output_Param55.DataSize = 1; Output_Param55.DataType = 'BYTE'; Output_Param56.Name = 'Output_Param56'; Output_Param56.HelpString = ''; Output_Param56.ReadOnly = False; Output_Param56.BitSize = 8; Output_Param56.DataSize = 1; Output_Param56.DataType = 'BYTE'; Output_Param57.Name = 'Output_Param57'; Output_Param57.HelpString = ''; Output_Param57.ReadOnly = False; Output_Param57.BitSize = 8; Output_Param57.DataSize = 1; Output_Param57.DataType = 'BYTE'; Output_Param58.Name = 'Output_Param58'; Output_Param58.HelpString = ''; Output_Param58.ReadOnly = False; Output_Param58.BitSize = 8; Output_Param58.DataSize = 1; Output_Param58.DataType = 'BYTE'; Output_Param59.Name = 'Output_Param59'; Output_Param59.HelpString = ''; Output_Param59.ReadOnly = False; Output_Param59.BitSize = 8; Output_Param59.DataSize = 1; Output_Param59.DataType = 'BYTE'; Output_Param60.Name = 'Output_Param60'; Output_Param60.HelpString = ''; Output_Param60.ReadOnly = False; Output_Param60.BitSize = 8; Output_Param60.DataSize = 1; Output_Param60.DataType = 'BYTE'; Output_Param61.Name = 'Output_Param61'; Output_Param61.HelpString = ''; Output_Param61.ReadOnly = False; Output_Param61.BitSize = 8; Output_Param61.DataSize = 1; Output_Param61.DataType = 'BYTE'; Output_Param62.Name = 'Output_Param62'; Output_Param62.HelpString = '';
              Output_Param62.ReadOnly = False; Output_Param62.BitSize = 8; Output_Param62.DataSize = 1; Output_Param62.DataType = 'BYTE'; Output_Param63.Name = 'Output_Param63'; Output_Param63.HelpString = ''; Output_Param63.ReadOnly = False; Output_Param63.BitSize = 8; Output_Param63.DataSize = 1; Output_Param63.DataType = 'BYTE'; ConfigVersion = 50660864
            unmapped channels: Input_Param0, Input_Param1, Input_Param2, Input_Param3, Input_Param4, Input_Param5, Input_Param6, Input_Param7, Input_Param8, Input_Param9, Input_Param10, Input_Param11, Input_Param12, Input_Param13, Input_Param14, Input_Param15, Input_Param16, Input_Param17, Input_Param18, Input_Param19, Input_Param20, Input_Param21, Input_Param22, Input_Param23, Input_Param24, Input_Param25, Input_Param26, Input_Param27, Input_Param28, Input_Param29, Input_Param30, Input_Param31, Input_Param32, Input_Param33, Input_Param34, Input_Param35, Input_Param36, Input_Param37, Input_Param38, Input_Param39,
              Input_Param40, Input_Param41, Input_Param42, Input_Param43, Input_Param44, Input_Param45, Input_Param46, Input_Param47, Input_Param48, Input_Param49, Input_Param50, Input_Param51, Input_Param52, Input_Param53, Input_Param54, Input_Param55, Input_Param56, Input_Param57, Input_Param58, Input_Param59, Input_Param60, Input_Param61, Input_Param62, Input_Param63, Output_Param0, Output_Param1, Output_Param2, Output_Param3, Output_Param4, Output_Param5, Output_Param6, Output_Param7, Output_Param8, Output_Param9, Output_Param10, Output_Param11, Output_Param12, Output_Param13, Output_Param14, Output_Param15,
              Output_Param16, Output_Param17, Output_Param18, Output_Param19, Output_Param20, Output_Param21, Output_Param22, Output_Param23, Output_Param24, Output_Param25, Output_Param26, Output_Param27, Output_Param28, Output_Param29, Output_Param30, Output_Param31, Output_Param32, Output_Param33, Output_Param34, Output_Param35, Output_Param36, Output_Param37, Output_Param38, Output_Param39, Output_Param40, Output_Param41, Output_Param42, Output_Param43, Output_Param44, Output_Param45, Output_Param46, Output_Param47, Output_Param48, Output_Param49, Output_Param50, Output_Param51, Output_Param52, Output_Param53, Output_Param54, Output_Param55,
              Output_Param56, Output_Param57, Output_Param58, Output_Param59, Output_Param60, Output_Param61, Output_Param62, Output_Param63
        VS_XXXX_Series : VS-XXXX Series, Keyence Corporation, order no. VS-XXXX Series , version Major Revision=16#1, Minor Revision = 16#1
            settings: INITIALIZED = TRUE; IP address of Target = [16#C0,16#A8,16#00,16#0A]; Keying.Check Minor Revision = FALSE; RequiredConfigVersion = 50660864; Number of Connections = 1; Connection Settings.Requested packet intervall = 10000 µs; Connection Settings.OT Connection Parameters = 18934; Connection Settings.TO Connection Parameters = 18502; Connection Settings.Connection Flags = 1056; Connection Settings.Connection Path Size = 8; Connection Settings.Large OT Connection Parameters = 1207960054; Connection Settings.Large TO Connection Parameters = 1207959622; Heartbeat Multiplier = 1; Trigger Ready.ReadOnly = False; Trigger Ready.BitSize = 1; Trigger Ready.DataSize = 1; Unused Parameter.ReadOnly = False; Unused Parameter.BitSize = 7; Unused Parameter.DataSize = 1; Trigger Ack.ReadOnly = False; Trigger Ack.BitSize = 1; Trigger Ack.DataSize = 1; Unused Parameter.ReadOnly = False; Unused Parameter.BitSize = 7; Unused Parameter.DataSize = 1; Pass.ReadOnly = False; Pass.BitSize = 1; Pass.DataSize = 1; Fail.ReadOnly = False; Fail.BitSize = 1; Fail.DataSize = 1; Unused Parameter.ReadOnly = False; Unused Parameter.BitSize = 1; Unused Parameter.DataSize = 1; Result Ready.ReadOnly = False; Result Ready.BitSize = 1; Result Ready.DataSize = 1; Run Status.ReadOnly = False; Run Status.BitSize = 1; Run Status.DataSize = 1;
              Unused Parameter.ReadOnly = False; Unused Parameter.BitSize = 1; Unused Parameter.DataSize = 1; Error0 Status.ReadOnly = False; Error0 Status.BitSize = 1; Error0 Status.DataSize = 1; Error1 Status.ReadOnly = False; Error1 Status.BitSize = 1; Error1 Status.DataSize = 1; Command Complete.ReadOnly = False; Command Complete.BitSize = 1; Command Complete.DataSize = 1; Command Error.ReadOnly = False; Command Error.BitSize = 1; Command Error.DataSize = 1; Command Ready.ReadOnly = False; Command Ready.BitSize = 1; Command Ready.DataSize = 1; Unused Parameter.ReadOnly = False; Unused Parameter.BitSize = 1; Unused Parameter.DataSize = 1; Program Load Complete.ReadOnly = False; Program Load Complete.BitSize = 1; Program Load Complete.DataSize = 1; Program Load Complete from SD Card.ReadOnly = False; Program Load Complete from SD Card.BitSize = 1; Program Load Complete from SD Card.DataSize = 1; Unused Parameter.ReadOnly = False; Unused Parameter.BitSize = 2; Unused Parameter.DataSize = 1; Soft Event 0 Ack.ReadOnly = False; Soft Event 0 Ack.BitSize = 1; Soft Event 0 Ack.DataSize = 1; Soft Event 1 Ack.ReadOnly = False; Soft Event 1 Ack.BitSize = 1; Soft Event 1 Ack.DataSize = 1; Soft Event 2 Ack.ReadOnly = False; Soft Event 2 Ack.BitSize = 1; Soft Event 2 Ack.DataSize = 1; Soft Event 3 Ack.ReadOnly = False;
              Soft Event 3 Ack.BitSize = 1; Soft Event 3 Ack.DataSize = 1; Soft Event 4 Ack.ReadOnly = False; Soft Event 4 Ack.BitSize = 1; Soft Event 4 Ack.DataSize = 1; Soft Event 5 Ack.ReadOnly = False; Soft Event 5 Ack.BitSize = 1; Soft Event 5 Ack.DataSize = 1; Soft Event 6 Ack.ReadOnly = False; Soft Event 6 Ack.BitSize = 1; Soft Event 6 Ack.DataSize = 1; Soft Event 7 Ack.ReadOnly = False; Soft Event 7 Ack.BitSize = 1; Soft Event 7 Ack.DataSize = 1; Assignable.ReadOnly = False; Assignable.BitSize = 24; Assignable.DataSize = 1; Tool Judge.ReadOnly = False; Tool Judge.BitSize = 32; Tool Judge.DataSize = 1; Error0 Code.ReadOnly = False; Error0 Code.BitSize = 32; Error0 Code.DataSize = 4; Error1 Code.ReadOnly = False; Error1 Code.BitSize = 32; Error1 Code.DataSize = 4; Program Number.ReadOnly = False; Program Number.BitSize = 32; Program Number.DataSize = 4; Total Count.ReadOnly = False; Total Count.BitSize = 32; Total Count.DataSize = 4; Result Data.ReadOnly = False; Result Data.BitSize = 32; Result Data.DataSize = 4; Result Data.ReadOnly = False; Result Data.BitSize = 32; Result Data.DataSize = 4; Result Data.ReadOnly = False; Result Data.BitSize = 32;
              Result Data.DataSize = 4; Result Data.ReadOnly = False; Result Data.BitSize = 32; Result Data.DataSize = 4; Result Data.ReadOnly = False; Result Data.BitSize = 32; Result Data.DataSize = 4; Result Data.ReadOnly = False; Result Data.BitSize = 32; Result Data.DataSize = 4; Result Data.ReadOnly = False; Result Data.BitSize = 32; Result Data.DataSize = 4; Result Data.ReadOnly = False; Result Data.BitSize = 32; Result Data.DataSize = 4; Result Data.ReadOnly = False; Result Data.BitSize = 32; Result Data.DataSize = 4; Result Data.ReadOnly = False; Result Data.BitSize = 32; Result Data.DataSize = 4; Trigger.ReadOnly = False; Trigger.BitSize = 1; Trigger.DataSize = 1; Unused Parameter.ReadOnly = False; Unused Parameter.BitSize = 7; Unused Parameter.DataSize = 1; Trigger Disable.ReadOnly = False; Trigger Disable.BitSize = 1; Trigger Disable.DataSize = 1; Output Disable.ReadOnly = False; Output Disable.BitSize = 1; Output Disable.DataSize = 1; Reset.ReadOnly = False; Reset.BitSize = 1; Reset.DataSize = 1; Unused Parameter.ReadOnly = False; Unused Parameter.BitSize = 5; Unused Parameter.DataSize = 1;
              Unused Parameter.ReadOnly = False; Unused Parameter.BitSize = 2; Unused Parameter.DataSize = 1; Result Handshake Enable.ReadOnly = False; Result Handshake Enable.BitSize = 1; Result Handshake Enable.DataSize = 1; Result Ack.ReadOnly = False; Result Ack.BitSize = 1; Result Ack.DataSize = 1; Go to Run.ReadOnly = False; Go to Run.BitSize = 1; Go to Run.DataSize = 1; Go to Setting.ReadOnly = False; Go to Setting.BitSize = 1; Go to Setting.DataSize = 1; Error0 Clear.ReadOnly = False; Error0 Clear.BitSize = 1; Error0 Clear.DataSize = 1; Error1 Clear.ReadOnly = False; Error1 Clear.BitSize = 1; Error1 Clear.DataSize = 1; Command Request.ReadOnly = False; Command Request.BitSize = 1; Command Request.DataSize = 1; Unused Parameter.ReadOnly = False; Unused Parameter.BitSize = 3; Unused Parameter.DataSize = 1; Program Load Execute.ReadOnly = False; Program Load Execute.BitSize = 1; Program Load Execute.DataSize = 1; Program Load Execute from SD Card.ReadOnly = False; Program Load Execute from SD Card.BitSize = 1; Program Load Execute from SD Card.DataSize = 1; Unused Parameter.ReadOnly = False; Unused Parameter.BitSize = 2; Unused Parameter.DataSize = 1; Soft Event 0.ReadOnly = False; Soft Event 0.BitSize = 1; Soft Event 0.DataSize = 1; Soft Event 1.ReadOnly = False;
              Soft Event 1.BitSize = 1; Soft Event 1.DataSize = 1; Soft Event 2.ReadOnly = False; Soft Event 2.BitSize = 1; Soft Event 2.DataSize = 1; Soft Event 3.ReadOnly = False; Soft Event 3.BitSize = 1; Soft Event 3.DataSize = 1; Soft Event 4.ReadOnly = False; Soft Event 4.BitSize = 1; Soft Event 4.DataSize = 1; Soft Event 5.ReadOnly = False; Soft Event 5.BitSize = 1; Soft Event 5.DataSize = 1; Soft Event 6.ReadOnly = False; Soft Event 6.BitSize = 1; Soft Event 6.DataSize = 1; Soft Event 7.ReadOnly = False; Soft Event 7.BitSize = 1; Soft Event 7.DataSize = 1; Assignable.ReadOnly = False; Assignable.BitSize = 24; Assignable.DataSize = 1; Program Number.ReadOnly = False; Program Number.BitSize = 32; Program Number.DataSize = 4; Parameter.ReadOnly = False; Parameter.BitSize = 3872; Parameter.DataSize = 4; Trigger Ready.Name = 'Trigger Ready'; Trigger Ready.HelpString = ''; Trigger Ready.ReadOnly = False; Trigger Ready.BitSize = 1; Trigger Ready.DataSize = 1; Unused Parameter.Name = 'Unused Parameter'; Unused Parameter.HelpString = ''; Unused Parameter.ReadOnly = False; Unused Parameter.BitSize = 7; Unused Parameter.DataSize = 1; Unused Parameter.DataType = 'BYTE';
              Trigger Ack.Name = 'Trigger Ack'; Trigger Ack.HelpString = ''; Trigger Ack.ReadOnly = False; Trigger Ack.BitSize = 1; Trigger Ack.DataSize = 1; Unused Parameter.Name = 'Unused Parameter'; Unused Parameter.HelpString = ''; Unused Parameter.ReadOnly = False; Unused Parameter.BitSize = 7; Unused Parameter.DataSize = 1; Unused Parameter.DataType = 'BYTE'; Pass.Name = 'Pass'; Pass.HelpString = ''; Pass.ReadOnly = False; Pass.BitSize = 1; Pass.DataSize = 1; Fail.Name = 'Fail'; Fail.HelpString = ''; Fail.ReadOnly = False; Fail.BitSize = 1; Fail.DataSize = 1; Unused Parameter.Name = 'Unused Parameter'; Unused Parameter.HelpString = ''; Unused Parameter.ReadOnly = False; Unused Parameter.BitSize = 1; Unused Parameter.DataSize = 1; Unused Parameter.DataType = 'BYTE'; Result Ready.Name = 'Result Ready'; Result Ready.HelpString = ''; Result Ready.ReadOnly = False; Result Ready.BitSize = 1; Result Ready.DataSize = 1; Run Status.Name = 'Run Status'; Run Status.HelpString = ''; Run Status.ReadOnly = False; Run Status.BitSize = 1; Run Status.DataSize = 1; Unused Parameter.Name = 'Unused Parameter'; Unused Parameter.HelpString = ''; Unused Parameter.ReadOnly = False;
              Unused Parameter.BitSize = 1; Unused Parameter.DataSize = 1; Unused Parameter.DataType = 'BYTE'; Error0 Status.Name = 'Error0 Status'; Error0 Status.HelpString = ''; Error0 Status.ReadOnly = False; Error0 Status.BitSize = 1; Error0 Status.DataSize = 1; Error1 Status.Name = 'Error1 Status'; Error1 Status.HelpString = ''; Error1 Status.ReadOnly = False; Error1 Status.BitSize = 1; Error1 Status.DataSize = 1; Command Complete.Name = 'Command Complete'; Command Complete.HelpString = ''; Command Complete.ReadOnly = False; Command Complete.BitSize = 1; Command Complete.DataSize = 1; Command Error.Name = 'Command Error'; Command Error.HelpString = ''; Command Error.ReadOnly = False; Command Error.BitSize = 1; Command Error.DataSize = 1; Command Ready.Name = 'Command Ready'; Command Ready.HelpString = ''; Command Ready.ReadOnly = False; Command Ready.BitSize = 1; Command Ready.DataSize = 1; Unused Parameter.Name = 'Unused Parameter'; Unused Parameter.HelpString = ''; Unused Parameter.ReadOnly = False; Unused Parameter.BitSize = 1; Unused Parameter.DataSize = 1; Unused Parameter.DataType = 'BYTE'; Program Load Complete.Name = 'Program Load Complete'; Program Load Complete.HelpString = ''; Program Load Complete.ReadOnly = False; Program Load Complete.BitSize = 1; Program Load Complete.DataSize = 1; Program Load Complete from SD Card.Name = 'Program Load Complete from SD Card';
              Program Load Complete from SD Card.HelpString = ''; Program Load Complete from SD Card.ReadOnly = False; Program Load Complete from SD Card.BitSize = 1; Program Load Complete from SD Card.DataSize = 1; Unused Parameter.Name = 'Unused Parameter'; Unused Parameter.HelpString = ''; Unused Parameter.ReadOnly = False; Unused Parameter.BitSize = 2; Unused Parameter.DataSize = 1; Unused Parameter.DataType = 'BYTE'; Soft Event 0 Ack.Name = 'Soft Event 0 Ack'; Soft Event 0 Ack.HelpString = ''; Soft Event 0 Ack.ReadOnly = False; Soft Event 0 Ack.BitSize = 1; Soft Event 0 Ack.DataSize = 1; Soft Event 1 Ack.Name = 'Soft Event 1 Ack'; Soft Event 1 Ack.HelpString = ''; Soft Event 1 Ack.ReadOnly = False; Soft Event 1 Ack.BitSize = 1; Soft Event 1 Ack.DataSize = 1; Soft Event 2 Ack.Name = 'Soft Event 2 Ack'; Soft Event 2 Ack.HelpString = ''; Soft Event 2 Ack.ReadOnly = False; Soft Event 2 Ack.BitSize = 1; Soft Event 2 Ack.DataSize = 1; Soft Event 3 Ack.Name = 'Soft Event 3 Ack'; Soft Event 3 Ack.HelpString = ''; Soft Event 3 Ack.ReadOnly = False; Soft Event 3 Ack.BitSize = 1; Soft Event 3 Ack.DataSize = 1; Soft Event 4 Ack.Name = 'Soft Event 4 Ack'; Soft Event 4 Ack.HelpString = ''; Soft Event 4 Ack.ReadOnly = False; Soft Event 4 Ack.BitSize = 1; Soft Event 4 Ack.DataSize = 1; Soft Event 5 Ack.Name = 'Soft Event 5 Ack'; Soft Event 5 Ack.HelpString = ''; Soft Event 5 Ack.ReadOnly = False; Soft Event 5 Ack.BitSize = 1; Soft Event 5 Ack.DataSize = 1;
              Soft Event 6 Ack.Name = 'Soft Event 6 Ack'; Soft Event 6 Ack.HelpString = ''; Soft Event 6 Ack.ReadOnly = False; Soft Event 6 Ack.BitSize = 1; Soft Event 6 Ack.DataSize = 1; Soft Event 7 Ack.Name = 'Soft Event 7 Ack'; Soft Event 7 Ack.HelpString = ''; Soft Event 7 Ack.ReadOnly = False; Soft Event 7 Ack.BitSize = 1; Soft Event 7 Ack.DataSize = 1; Assignable.Name = 'Assignable'; Assignable.HelpString = ''; Assignable.ReadOnly = False; Assignable.BitSize = 24; Assignable.DataSize = 1; Tool Judge.Name = 'Tool Judge'; Tool Judge.HelpString = ''; Tool Judge.ReadOnly = False; Tool Judge.BitSize = 32; Tool Judge.DataSize = 1; Error0 Code.Name = 'Error0 Code'; Error0 Code.HelpString = ''; Error0 Code.ReadOnly = False; Error0 Code.BitSize = 32; Error0 Code.DataSize = 4; Error0 Code.DataType = 'UDINT'; Error1 Code.Name = 'Error1 Code'; Error1 Code.HelpString = ''; Error1 Code.ReadOnly = False; Error1 Code.BitSize = 32; Error1 Code.DataSize = 4; Error1 Code.DataType = 'UDINT'; Program Number.Name = 'Program Number'; Program Number.HelpString = ''; Program Number.ReadOnly = False; Program Number.BitSize = 32; Program Number.DataSize = 4; Program Number.DataType = 'UDINT'; Total Count.Name = 'Total Count'; Total Count.HelpString = '';
              Total Count.ReadOnly = False; Total Count.BitSize = 32; Total Count.DataSize = 4; Total Count.DataType = 'UDINT'; Result Data.Name = 'Result Data'; Result Data.HelpString = ''; Result Data.ReadOnly = False; Result Data.BitSize = 32; Result Data.DataSize = 4; Result Data.DataType = 'UDINT'; Result Data.Name = 'Result Data'; Result Data.HelpString = ''; Result Data.ReadOnly = False; Result Data.BitSize = 32; Result Data.DataSize = 4; Result Data.DataType = 'UDINT'; Result Data.Name = 'Result Data'; Result Data.HelpString = ''; Result Data.ReadOnly = False; Result Data.BitSize = 32; Result Data.DataSize = 4; Result Data.DataType = 'UDINT'; Result Data.Name = 'Result Data'; Result Data.HelpString = ''; Result Data.ReadOnly = False; Result Data.BitSize = 32; Result Data.DataSize = 4; Result Data.DataType = 'UDINT'; Result Data.Name = 'Result Data'; Result Data.HelpString = ''; Result Data.ReadOnly = False; Result Data.BitSize = 32; Result Data.DataSize = 4; Result Data.DataType = 'UDINT'; Result Data.Name = 'Result Data'; Result Data.HelpString = ''; Result Data.ReadOnly = False; Result Data.BitSize = 32; Result Data.DataSize = 4; Result Data.DataType = 'UDINT';
              Result Data.Name = 'Result Data'; Result Data.HelpString = ''; Result Data.ReadOnly = False; Result Data.BitSize = 32; Result Data.DataSize = 4; Result Data.DataType = 'UDINT'; Result Data.Name = 'Result Data'; Result Data.HelpString = ''; Result Data.ReadOnly = False; Result Data.BitSize = 32; Result Data.DataSize = 4; Result Data.DataType = 'UDINT'; Result Data.Name = 'Result Data'; Result Data.HelpString = ''; Result Data.ReadOnly = False; Result Data.BitSize = 32; Result Data.DataSize = 4; Result Data.DataType = 'REAL'; Result Data.Name = 'Result Data'; Result Data.HelpString = ''; Result Data.ReadOnly = False; Result Data.BitSize = 32; Result Data.DataSize = 4; Result Data.DataType = 'REAL'; Trigger.Name = 'Trigger'; Trigger.HelpString = ''; Trigger.ReadOnly = False; Trigger.BitSize = 1; Trigger.DataSize = 1; Unused Parameter.Name = 'Unused Parameter'; Unused Parameter.HelpString = ''; Unused Parameter.ReadOnly = False; Unused Parameter.BitSize = 7; Unused Parameter.DataSize = 1; Unused Parameter.DataType = 'BYTE'; Trigger Disable.Name = 'Trigger Disable'; Trigger Disable.HelpString = ''; Trigger Disable.ReadOnly = False; Trigger Disable.BitSize = 1; Trigger Disable.DataSize = 1;
              Output Disable.Name = 'Output Disable'; Output Disable.HelpString = ''; Output Disable.ReadOnly = False; Output Disable.BitSize = 1; Output Disable.DataSize = 1; Reset.Name = 'Reset'; Reset.HelpString = ''; Reset.ReadOnly = False; Reset.BitSize = 1; Reset.DataSize = 1; Unused Parameter.Name = 'Unused Parameter'; Unused Parameter.HelpString = ''; Unused Parameter.ReadOnly = False; Unused Parameter.BitSize = 5; Unused Parameter.DataSize = 1; Unused Parameter.DataType = 'BYTE'; Unused Parameter.Name = 'Unused Parameter'; Unused Parameter.HelpString = ''; Unused Parameter.ReadOnly = False; Unused Parameter.BitSize = 2; Unused Parameter.DataSize = 1; Unused Parameter.DataType = 'BYTE'; Result Handshake Enable.Name = 'Result Handshake Enable'; Result Handshake Enable.HelpString = ''; Result Handshake Enable.ReadOnly = False; Result Handshake Enable.BitSize = 1; Result Handshake Enable.DataSize = 1; Result Ack.Name = 'Result Ack'; Result Ack.HelpString = ''; Result Ack.ReadOnly = False; Result Ack.BitSize = 1; Result Ack.DataSize = 1; Go to Run.Name = 'Go to Run'; Go to Run.HelpString = ''; Go to Run.ReadOnly = False; Go to Run.BitSize = 1; Go to Run.DataSize = 1; Go to Setting.Name = 'Go to Setting'; Go to Setting.HelpString = ''; Go to Setting.ReadOnly = False;
              Go to Setting.BitSize = 1; Go to Setting.DataSize = 1; Error0 Clear.Name = 'Error0 Clear'; Error0 Clear.HelpString = ''; Error0 Clear.ReadOnly = False; Error0 Clear.BitSize = 1; Error0 Clear.DataSize = 1; Error1 Clear.Name = 'Error1 Clear'; Error1 Clear.HelpString = ''; Error1 Clear.ReadOnly = False; Error1 Clear.BitSize = 1; Error1 Clear.DataSize = 1; Command Request.Name = 'Command Request'; Command Request.HelpString = ''; Command Request.ReadOnly = False; Command Request.BitSize = 1; Command Request.DataSize = 1; Unused Parameter.Name = 'Unused Parameter'; Unused Parameter.HelpString = ''; Unused Parameter.ReadOnly = False; Unused Parameter.BitSize = 3; Unused Parameter.DataSize = 1; Unused Parameter.DataType = 'BYTE'; Program Load Execute.Name = 'Program Load Execute'; Program Load Execute.HelpString = ''; Program Load Execute.ReadOnly = False; Program Load Execute.BitSize = 1; Program Load Execute.DataSize = 1; Program Load Execute from SD Card.Name = 'Program Load Execute from SD Card'; Program Load Execute from SD Card.HelpString = ''; Program Load Execute from SD Card.ReadOnly = False; Program Load Execute from SD Card.BitSize = 1; Program Load Execute from SD Card.DataSize = 1; Unused Parameter.Name = 'Unused Parameter'; Unused Parameter.HelpString = ''; Unused Parameter.ReadOnly = False; Unused Parameter.BitSize = 2; Unused Parameter.DataSize = 1; Unused Parameter.DataType = 'BYTE'; Soft Event 0.Name = 'Soft Event 0';
              Soft Event 0.HelpString = ''; Soft Event 0.ReadOnly = False; Soft Event 0.BitSize = 1; Soft Event 0.DataSize = 1; Soft Event 1.Name = 'Soft Event 1'; Soft Event 1.HelpString = ''; Soft Event 1.ReadOnly = False; Soft Event 1.BitSize = 1; Soft Event 1.DataSize = 1; Soft Event 2.Name = 'Soft Event 2'; Soft Event 2.HelpString = ''; Soft Event 2.ReadOnly = False; Soft Event 2.BitSize = 1; Soft Event 2.DataSize = 1; Soft Event 3.Name = 'Soft Event 3'; Soft Event 3.HelpString = ''; Soft Event 3.ReadOnly = False; Soft Event 3.BitSize = 1; Soft Event 3.DataSize = 1; Soft Event 4.Name = 'Soft Event 4'; Soft Event 4.HelpString = ''; Soft Event 4.ReadOnly = False; Soft Event 4.BitSize = 1; Soft Event 4.DataSize = 1; Soft Event 5.Name = 'Soft Event 5'; Soft Event 5.HelpString = ''; Soft Event 5.ReadOnly = False; Soft Event 5.BitSize = 1; Soft Event 5.DataSize = 1; Soft Event 6.Name = 'Soft Event 6'; Soft Event 6.HelpString = ''; Soft Event 6.ReadOnly = False; Soft Event 6.BitSize = 1; Soft Event 6.DataSize = 1; Soft Event 7.Name = 'Soft Event 7'; Soft Event 7.HelpString = ''; Soft Event 7.ReadOnly = False; Soft Event 7.BitSize = 1; Soft Event 7.DataSize = 1; Assignable.Name = 'Assignable';
              Assignable.HelpString = ''; Assignable.ReadOnly = False; Assignable.BitSize = 24; Assignable.DataSize = 1; Program Number.Name = 'Program Number'; Program Number.HelpString = ''; Program Number.ReadOnly = False; Program Number.BitSize = 32; Program Number.DataSize = 4; Program Number.DataType = 'UDINT'; Parameter.Name = 'Parameter'; Parameter.HelpString = ''; Parameter.ReadOnly = False; Parameter.BitSize = 3872; Parameter.DataSize = 4; Parameter.DataType = 'UDINT'; ConfigVersion = 50660864
            input  Application.GVL.CAM_1.TRIGGER_READY : BOOL  // Trigger Ready
            input  Application.GVL.CAM_1.RESULTS_READY : BOOL  // Result Ready
            input  Application.GVL.CAM_1.CURRENT_COUNT : UDINT  // Total Count
            input  Application.GVL.CAM_1.Result_Count : UDINT  // Result Data
            input  Application.GVL.CAM_1.Result_PosX : REAL  // Result Data
            input  Application.GVL.CAM_1.Result_PosY : REAL  // Result Data
            output Application.GVL.CAM_1.Trigger : BOOL  // Trigger
            unmapped channels: Unused Parameter, Trigger Ack, Unused Parameter, Pass, Fail, Unused Parameter, Run Status, Unused Parameter, Error0 Status, Error1 Status, Command Complete, Command Error, Command Ready, Unused Parameter, Program Load Complete, Program Load Complete from SD Card, Unused Parameter, Soft Event 0 Ack, Soft Event 1 Ack, Soft Event 2 Ack, Soft Event 3 Ack, Soft Event 4 Ack, Soft Event 5 Ack, Soft Event 6 Ack, Soft Event 7 Ack, Assignable, Tool Judge, Error0 Code, Error1 Code, Program Number, Result Data, Result Data, Result Data, Result Data, Result Data, Result Data, Result Data, Unused Parameter, Trigger Disable, Output Disable,
              Reset, Unused Parameter, Unused Parameter, Result Handshake Enable, Result Ack, Go to Run, Go to Setting, Error0 Clear, Error1 Clear, Command Request, Unused Parameter, Program Load Execute, Program Load Execute from SD Card, Unused Parameter, Soft Event 0, Soft Event 1, Soft Event 2, Soft Event 3, Soft Event 4, Soft Event 5, Soft Event 6, Soft Event 7, Assignable, Program Number, Parameter
  libraries: VisuSymbols, 4.5.0.0 (System)
  text list GlobalTextList
*)

// Device/Application/F1000_UDTs/E_SchedState
TYPE E_SchedState :
(
    INIT,
    WAIT_FOR_START,
    RUN_FORWARD,
    DELAY_BETWEEN,
    RUN_REVERSE,
    DONE
);
END_TYPE

// Device/Application/F1000_UDTs/UDT_Explicit
TYPE UDT_Explicit :
STRUCT
	xTriggerWrite: BOOL;
	xWriteDone: BOOL;
	xWriteBusy: BOOL;
	xWriteError: BOOL;
	eWriteErrorCode: ENIP.Error;
END_STRUCT
END_TYPE

// Device/Application/F1000_UDTs/UDT_PARTX
TYPE UDT_PARTX :
STRUCT
	IP_ADDR: STRING(16):='192.168.1.11';
	ENABLE_TCP:BOOL;
	Amp1: BYTE;
	Amp2: BYTE;
	Amp3: BYTE;
	Amp4: BYTE;
	Freq: BYTE;
	BackLight:BOOL;
	Feeder_Enable:BOOL;
	FWD:BOOL;
	BACK:BOOL;
	SHAKE:BOOL;
	MAN:BOOL;
	
	
END_STRUCT
END_TYPE

// Device/Application/F1000_UDTs/UDT_Robot
TYPE UDT_Robot :
STRUCT
	Test: REAL;
END_STRUCT
END_TYPE

// Device/Application/F1000_UDTs/UDT_StepConfig
TYPE UDT_StepConfig :
STRUCT
	StepEnable : BOOL;  // The "ON" checkbox
	Direction  : INT;   // 0 = None, 1 = FWD/UP, 2 = REV/DOWN (Dropdown link)
	DurationMS : DINT := 1000; // Duration in milliseconds from the HMI numbox
END_STRUCT
END_TYPE

// Device/Application/F1000_UDTs/UDT_SYS
TYPE UDT_SYS :
STRUCT
	STEP: DINT;
	STEP_IMG: DINT;
	CYCLE_START: BOOL;
	CYCLE_STOP: BOOL;
	RESET:BOOL;
	CONTROL_ON:BOOL;
	SET_TRF:BOOL;
	RBT_ERROR: GetErrors;
	HOME_RBT:BOOL;
	
	
END_STRUCT
END_TYPE

// Device/Application/F1000_UDTs/UDT_VS_Series
TYPE UDT_VS_Series :
STRUCT
	RESULT_POSX: REAL;
	RESULT_POSY: REAL;
	RESULT_COUNT: UDINT;
	TRIGGER: BOOL;
	TRIGGER_READY: BOOL;
	RESULTS_READY:BOOL;
	OLD_COUNT: DINT;
	CURRENT_COUNT:DINT;
	
END_STRUCT
END_TYPE

// Device/Application/F1000_UDTs/UDT_Meca500/ENUM/Meca500_DynamicDataTypeID
{attribute 'qualified_only'}
{attribute 'strict'}
///For more informations refer to page 75 of the documentation meca500-r4-programming-manual.
TYPE Meca500_DynamicDataTypeID :
(
	///Robot will automatically choose dynamic data type and change it every cycle to go through
	///them all. This is the easiest way for the host to receive all possible values periodically (round-robin
	///manner).
	AUTOMATIC:=0,
	
	///Firmware version. Values: [major version, minor version, patch version, build number]. Same as
	///GetFwVersion.
	FIRMWARE_VERSION:=1,
	
	///Product type. Values: [product type (3=Meca500)]. Same as GetProductType.
	PRODUCT_TYPE:=2,
	
	///Serial number. Values: [serial number]. Same as GetRobotSerial.
	SERIAL_NUMBER:=3,
	
	///Joints offset (as calculated by mastering at production). Values: [δθ1, δθ2, δθ3, δθ4, δθ5, δθ6]. In degrees.
	GET_JOINTS_OFFSET:=4,
	
	///Joint limits enabled state. Values: [enabled 1/0]. Same as GetJointLimitsCfg.
	GET_JOINT_LIMITS_CFG:=11,
	
	///Robot model's nominal joint limits for joints 1, 2 and 3. Values: [θ1,min, θ1,max, θ2,min, θ2,max, θ3,min, θ3,max].
	///Unit is degrees. Same as GetModelJointLimits.
	GET_MODEL_JOINT_1_TO_3_LIMITS:=12,
	
	///Robot model's nominal joint limits for joints 4, 5 and 6. Values: [θ4,min, θ4,max, θ5,min, θ5,max, θ6,min, θ6,max].
	///Unit is degrees. Same as GetModelJointLimits.
	GET_MODEL_JOINT_4_TO_6_LIMITS:=13,
	
	///Effective joint limits for joints 1, 2 and 3. Values: [θ1,min, θ1,max, θ2,min, θ2,max, θ3,min, θ3,max]. Unit is degrees.
	///Same as GetJointLimits.
	GET_EFF_JOINT_1_to_3_LIMITS:=14,
	
	///Effective joint limits for joints 4, 5 and 6. Values: [θ4,min, θ4,max, θ5,min, θ5,max, θ6,min, θ6,max]. Unit is degrees.
	///Same as GetJointLimits.
	GET_EFF_JOINT_4_TO_6_LIMITS:=15,
	
	///Current workspace limits configuration. Values: [workspace limits severity, workspace limits detection mode].
	///Same as GetWorkspaceLimitsCfg.
	GET_WORKSPACE_LIMITS_CFG:=17,
	
	///Current workspace Limits. Values: [xmin, ymin, zmin, xmax, ymax, zmax]. Units is mm. Same as
	///GetWorkspaceLimits.
	GET_WORKSPACE_LIMITS:=18,
	
	///Tool Sphere model. Values: [x, y, z, r]. Units in mm. Same as GetToolSphere.
	GET_EFF_TOOL_SPHERE:=19,
	
	///Motion queue's conf that will be applied to next MovePose. Values: [shoulder −1/1/NaN, elbow −1/1/NaN,
	///wrist −1/1/NaN, last joint turn or NaN]. Value NaN is used to indicate auto-conf or auto-conf-turn. Same as
	///GetConf and GetConfTurn.
	GET_MOTION_QUEUE_CONF:=20,
	
	///Motion queue parameters. Values: [blending ratio percent, velocity timeout in seconds]. Same as
	///GetBlending AND GetVelTimeout.
	GET_MOTION_QUEUE_PARAM:=21,
	
	///Motion queue velocities and accelerations in percent. Values: [joint velocity, joint acceleration, Cartesian
	///linear velocity, Cartesian angular velocity, Cartesian acceleration]. Unit is percent. Same as GetJointVel,
	///GetJointAcc, GetCartLinVel, GetCartAngVel, and GetCartAcc.
	GET_MOTION_PARAM:=22,
	
	///Gripper parameters. Values: [gripper force, gripper velocity, fingers opening corresponding to closed state,
	///fingers opening corresponding to open state]. Arguments 1 and 2 are in percentage, while arguments 3
	///and 4 are in mm. Same as GetGripperForce, GetGripperVel, and GetGripperRange.
	GET_GRIPPER_PARAM:=23,
	
	///Torque limits configuration. Values: [severity, detection mode]. See Section 2.1.28 of programming manual for corresponding
	///severity/mode values. Same as GetTorqueLimitsCfg.
	GET_TORQUE_LIMITS_CFG:=24,
	
	///Torque limits. Values: [joint 1 limit, joint 2 limit, ..., joint 6 limit]. Unit is percent. Same as GetTorqueLimits.
	GET_TORQUE_LIMITS:=25,
	
	///Target real-time joint velocity. Values: [θ̇ 1, θ̇ 2, θ̇ 3, θ̇ 4, θ̇ 5, θ̇ 6]. Unit is °/s. Same as GetRtTargetJointVel.
	GET_RT_TARET_JOINT_VEL:=32,
	
	///Target real-time joint torque (not implemented yet). Values: [joint 1 torque, joint 2 torque, ..., joint 6
	///torque]. Unit is percent. Same as GetRtTargetJointTorq.
	GET_RT_TARGET_JOINT_TORQ:=33,
	
	///Target real-time Cartesian velocity (TRF with respect to. WRF). Values: [ẋ , ẏ , ż, ωx, ωy, ωz]. Units are mm/s
	///or °/s. Same as GetRtTargetCartVel.
	GET_RT_TARGET_CART_VEL:=34,
	
	///Actual real-time joint position based on hardware encoders. Values: [θ1, θ2, θ3, θ4, θ5, θ6]. Unit is degrees.
	///Same as GetRtJointPos.
	GET_RT_JOINT_POS:=40,
	
	///Actual real-time end-effector pose (TRF with respect to. WRF). Values: [x, y, z, α, β, γ]. Units are mm or
	///degrees. Same as GetRtCartPos.
	GET_RT_CART_POS:=41,
	
	///Actual real-time joint velocity. Values: [θ̇ 1, θ̇ 2, θ̇ 3, θ̇ 4, θ̇ 5, θ̇6]. Unit is °/s. Same as GetRtJointVel.	
	GET_RT_JOINT_VEL:=42,
	
	///Actual REAL-TIME joint torque. Values: [joint 1 torque, joint 2 torque, ..., joint 6 torque]. Unit is percent.
	///Same as GetRtJointTorq.
	GET_RT_JOINT_TORQ:=43,
	
	///Actual real-time cartesian velocity (TRF with respect to. WRF). Values: [ẋ , ẏ , ż, ωx, ωy, ωz]. Units are mm/s
	///or °/s. Same as GetRtCartVel.
	GET_RT_CART_VEL:=44,
	
	///Actual conf that corresponds to real-time end-effector pose. Values: [shoulder −1/0/1, elbow −1/0/1, 
	///wrist−1/0/1, last joint turn]. Same as GetRtConf and GetRtConfTurn.
	GET_RT_CONF:=45,
	
	///Accelerometer reading. Values: [ax, ay, az]. Unit is 1/16,000 of G. Same as GetRtAccelerometer.
	GET_RT_ACCELOMETER:=46,
	
	///External tool status. Values: [type, homing done, error state, overheated]. Same as GetRtExtToolStatus.
	GET_RT_EXT_TOOL_STATUS:=52,
	
	///EOAT status. Values if type gripper: [holding part, desired fingers opening reached, gripper closed, gripper
	///open, gripper force, fingers opening]. Values if pneumatic module: [valve 1 state, valve 2 state].
	GET_EOT_STATUS:=53

);
END_TYPE

// Device/Application/F1000_UDTs/UDT_Meca500/ENUM/Meca500_Errors
{attribute 'qualified_only'}
{attribute 'strict'}
///For more informations refer to page 52 of the documentation meca500-r4-programming-manual.
TYPE Meca500_Errors :
(
	 ///No error currently.
	 NO_ERROR := 0,
	
	 ///Maximum number OF queued commands reached. Retry BY sending commands AT a slower rate.
	 COMMAND_BUFFER_IS_FULL := 1000,
	
	 ///Unknown or empty command.
	 UNKNOWN_COMMAND := 1001,
	
	 ///Syntax error or symbol missing. - Command: '...'] A parenthesis or a comma has been omitted.
	 SYNTAX_ERROR := 1002, 
	
	 ///Wrong number of arguments or invalid input (e.g., the argument is out of range).
	 ARGUMENT_ERROR := 1003,
	
	 ///The robot must be activated.
	 THE_ROBOT_IS_NOT_ACTIVATED := 1005,
	
	 ///The robot must be homed.
	 THE_ROBOT_IS_NOT_HOMED := 1006,
	
	 ///The robot cannot reach the joint set or pose requested because of its joint limits.
	 JOINT_OVER_LIMIT := 1007, 
	 
	 ///The linear motion cannot be executed because it requires a reorientation of 180° of the end-effector,
	 ///and there may be two possible paths.
	 SINGULARITY_DETECTED_ROTATE:=1010,
	
	 ///A command has been sent but the robot is in error mode and cannot process it until a ResetError command is sent.
	 THE_ROBOT_IS_IN_ERROR := 1011,
	
	 ///The MoveLin command sent requires that the robot pass through a singularity, or the MovePose command sent requires that the robot goes to a singular robot posture.
	 SINGULARITY_DETECTED_REORIENTATION := 1012,
	
	 ///Activation failed. Try again. 
	 ACTIVATION_FAILED := 1013,
	
	 ///Homing procedure failed. Try again.
	 HOMING_FAILED := 1014,
	
	 ///The pose requested in the MoveLin or MovePose commands cannot be reached by the robot (even if the robot had no joint limits).
	 POSE_OUT_OF_REACH := 1016,
	
	 ///Problem with communication.
	 COMMUNICATION_FAILED := 1017,
	
	 ///Missing NULL character at the end of a command.
	 MISSING_NULL := 1018,
	
	 ///Something is wrong. The brakes cannot be engaged. Try again.
	 BRAKES_CANNOT_BE_RELEASED := 1020,
	
	 ///Something is wrong. The deactivation failed. Try again.
	 DEACTIVATION_FAILED := 1021,
	
	 ///The command StopSaving was sent, but the robot was not saving a program.
	 PROGRAM_SAVING_FAILED_1 := 1022,
	
	 ///The command cannot be executed in the offline program.
	 IGNORING_COMMAND_FOR_OFFLINE_MODE := 1023,
	
	 ///Somehow, mastering was lost. Contact Mecademic.
	 MASTERING_NEEDED := 1024,
	
	 ///Turn off the robot, then turn it back on in order to reset the error.
	 RESET_ERROR_NOT_POSSIBLE := 1025, 
	
	 ///The robot must be deactivated in order to execute this command.
	 DEACTIVATION_NEEDED := 1026,
	
	 ///The robot must be deactivated in order to execute this command.
	 CHANGE_SIMULATION_MODE_FAILED := 1027,
	
	 ///Error on the network. Resend the command.
	 NETWORK_ERROR := 1028,
	
	 ///Maximum program size is 13,000 commands. Saving stopped - Memory full.
	 OFFLINE_PROGRAM_FULL := 1029,
	
	 ///The robot is already saving a program. Wait until finished to save another program.
	 ALREADY_SAVING := 1030,
	
	 ///The command cannot be executed because the robot is currently saving a program.
	 PROGRAM_SAVING_ABORTED := 1031,
	 
	 ///Requested move blocked because start robot position is not in the requested configuration.
	 START_CONF_MISMATCH := 1033,
	
	 ///No gripper was detected.
	 ERR_NO_GRIPPER_CONNECTED := 1038,
	 
	 ///General error for various commands.
	 COMMAND_FAILED := 1040,
	 
	 ///No pneumatic model connected.
	 NO_VBOX := 1041,
	 
	 ///Switching external tool type is only possible when the robot is deactivated.
	 EXT_TOOL_SIM_MUST_DEACT := 1042,
	
	  ///If the gripper was forcing when this message appeared, most probably an overheating occurred. 
	 ///Let the gripper cool down for a few minutes and send the ResetError command. 
	 ///Note that the gripper will stop applying a force, so if it was holding a part, the part might fall.
	 GRIPPER_ERROR := 3025,
	 
	 ///A hardware problem was detected. Mecademic cannot guaranty correct movements - Please contact Mecademic.
	 MAINTENANCE_CHECK_DISCOVERED_A_PROBLEM := 3026,
	 
	 ///A communication error with the pneumatic module was detected. Contact Mecademic.
	 PNEUMATIC_ERROR := 3037
);
END_TYPE

// Device/Application/F1000_UDTs/UDT_Meca500/ENUM/Meca500_MotionCommandID
{attribute 'qualified_only'}
{attribute 'strict'}
/// For more information refer to page 72 of the documentation meca500-r4-programming-manual
TYPE Meca500_MotionCommandID :
(
	 /// No Motion command active
	 NO_COMMAND := 0,
	  
	 /// This command makes the robot rotate simultaneously its joints to the specified joint set. 
	 /// All joint rotations start and stop at the same time. The path that the robot takes is linear in
	 /// the joint space, but nonlinear in the Cartesian space. Therefore, the TCP trajectory is not
	 /// easily predictable. Finally, with MoveJoints, the robot can cross singularities.
	 /// All six subindices are in degrees.
	 MOVE_JOINTS := 1,
	  
	 /// This command makes the robot move its TRF to a specific pose with respect TO the WRF.
	 /// Essentially, the robot controller calculates all possible joint sets corresponding to the desired
	 /// pose and for which euler angle 6 is in the range +/-180°, except those corresponding to a singular robot
	 /// posture. Then, it either chooses the joint set that corresponds to the desired configuration guration or
	 /// the one that is fastest to reach (see SetConf and SetAutoConf). Finally, it executes internally
	 /// a MoveJoints command with the chosen joint set.
	 /// Thus, all joint rotations start and stop at the same time. The path the robot takes is
	 /// linear in the joint-space, but nonlinear in Cartesian space. Therefore, the path the TCP will
	 /// follow to its final destination is not easily predictable, as illustrated in Fig. 7.
	 /// Using this command, the robot can cross a singularity or start from a singular robot
	 /// posture, as long as SetAutoConf is enabled. However, the robot cannot go to a singular robot
	 /// posture using MovePose. For example, assuming that the TRF coincides with the FRF, you
     /// cannot execute the command MovePose(190,0,308,0,90,0), since this pose corresponds only
	 /// to singular robot posture (e.g., the joint set {0,0,0,0,0,0}). You can only use the MovePose
	 /// command with a pose that corresponds to at least one non-singular robot posture.
	 /// As with the MoveJoints command, if the complete motion cannot be performed due to
     /// singularities or joint limits, it will normally not even start, and an error will be generated.
     /// Finally, note that this command will make the robot move to a joint set (corresponding
	 /// to the desired pose) for which euler angle 6 is in the range +/-180°. Finally, note that this command will
	 /// be executed only if euler angle 6 is already in the range +/-180°.  
	 /// Subindices 1, 2, 3 are in mm and 4, 5, 6 are in degrees.
	 MOVE_POSE := 2,
	  
	 /// This command makes the robot move its TRF to a specific pose with respect to the WRF
	 /// while keeping the TCP along a linear path in Cartesian space, as illustrated in Fig. 8. If the
	 /// final (desired) orientation of the TRF is different from the initial orientation, the orientation
	 /// will be modified along the path using LERP interpolation.
	 /// Using this command, the robot cannot move to or through a singular robot posture or one
	 /// that is too close to being singular. This command cannot automatically change the robot
	 /// configuration. Furthermore, note that when executing this command, euler angle 6 must already be in
	 /// the the range +/-180° and will remain in that range during the execution of the command.
	 /// Finally, note that if the motion requires that a joint rotates more than 180°, it will not be
	 /// executed (unless you are upgrading from firmware 7). Furthermore, if the complete motion
	 /// cannot be performed due to singularities or joint limits, it will normally not even start, and
	 /// an error will be generated.
	 /// Subindices 1, 2, 3 are in mm and 4, 5, 6 are in degrees.  
	 MOVE_LIN := 3, 
	  
	 /// This command is similar to the MoveLin command, but allows a desired pose to be specified
	 /// relative to the current pose of the TRF. Thus, the arguments X, Y, Z, Rx, Ry, Rz represent the
	 /// desired pose of the TRF with respect to the current pose of the TRF (i.e., the pose of the
	 /// TRF just before executing the MoveLinRelTRF command).
	 /// As with the MoveLin command, if the complete motion cannot be performed due to
	 /// singularities or joint limits, it will normally not even start and an error will be generated.
	 /// These joint limits include the fact that joint 6 must be in the range +/-180° at all times and
	 /// no joint can rotate more than 180° (in a single linear displacement).
	 /// Subindices 1, 2, 3 are in mm and 4, 5, 6 are in degrees.
	 MOVE_LIN_REL_TRF := 4,
	  
	 /// This command is similar to the MoveLinRelTRF command, but instead of defening the
	 /// desired pose with respect to the current pose of the TRF it is defined with respect to a
	 /// reference frame that has the same orientation as the WRF but its origin is at the current
	 /// position of the TCP.
	 /// As with the MoveLin command, if the complete motion cannot be performed due to
	 /// singularities or joint limits, it will not even start. These joint limits include the fact that
	 /// joint 6 must be in the range +/-180° at all times and no joint can rotate more than 180° (in
	 /// a single linear displacement).
	 /// Subindices 1, 2, 3 are in mm and 4, 5, 6 are in degrees. 
	 MOVE_LIN_REL_WRF := 5,
	  
	 /// This command is used to add a time delay after a motion command. In other words, the
	 /// robot completes all movements sent before the Delay command and stops temporarily. (In
	 /// contrast, the PauseMotion command interrupts the motion as soon as received by the robot.)
	 /// Subindex 1 is the pause in seconds. 
	 DELAY := 6,
	  
	 /// This command enables/disables the robot's blending feature (recall Section 2.2.2). Note
	 /// that the commands MoveLin, MovePose, and MoveJoints will only send "[3004][End of move-
	 /// ment.]" responses when the robot comes to a complete stop and the command SetEOM(1)
	 /// was used. Therefore, enabling blending may suppress these responses.
	 /// Also, note that there is blending only between consecutive movements with the commands
	 /// MoveJoints and MovePose, or between consecutive movements with the commands MoveLin,
	 /// MoveLinRelTRF and MoveLinRelTRF. In other words, there will never be blending between
	 /// the trajectories of a MovePose command followed by a MoveLin command. 
	 /// Subindex 1 is the percentage of blending, from 0 or 100.
	 SET_BLENDING := 7,
	  
	 /// This command limits the angular velocities of the robot joints. It affects the movements
	 /// generated by the MovePose and MoveJoints commands.
	 /// It is not possible to limit the velocity of only one joint. With this command, the maximum
	 /// velocities of all joints are limited proportionally. The maximum velocity of each joint will
	 /// be reduced to a percentage p of its top velocity. The top velocity of joints 1 and 2 is 150°/s,
	 /// of joint 3 is 180°/s, of joints 4 and 5 is 300°/s, and of joint 6 is 500°/s.
	 /// Subindex 1 is the percentage of maximum joint velocities, from 0.001 to 100.
	 SET_JOINT_VEL := 8,
	  
	 /// This command limits the acceleration of the joints during movements resulting from joint-
	 /// space commands (see Fig. 6). Note that this command makes the robot stop, even if blending
	 /// is enabled.
	 /// Note that the argument of this command is exceptionally limited to 150. This is because
	 /// in firmware 8, a scaling was applied so that if this argument is kept at 100, most joint-
	 /// space movements are feasible even at full payload. More precisely, if you are upgrading from
	 /// firmware 7 and you want to keep the same joint accelerations, you need to multiply the
	 /// arguments of your SetJointAcc commands by the factor 1.43.
	 /// Subindex 1 is the percentage of maximum joint accelerations, from 0.001 to 150.
	 SET_JOINT_ACC := 9,
	  
	 /// This command limits the angular velocity of the robot TRF with respect to its WRF. It only
	 /// affects the movements generated by the MoveLin, MoveLinRelTRF and MoveLinRelWRF
	 /// commands.
	 /// Subindex 1 is the Cartesian angular velocity limit, from 0.001 to 300, measured in °/s.
	 SET_CART_ANG_VEL := 10,
	 
	 /// This command limits the Cartesian linear velocity of the robot's TRF with respect to
	 /// its WRF. It only affects the movements generated by the MoveLin, MoveLinRelTRF and
	 /// MoveLinRelWRF commands.
	 /// Subindex 1 is the linear velocity limit for the TCP, from 0.001 to 1,000, measured in mm/s.
	 SET_CART_LIN_VEL := 11, 
	  
	 /// This command limits the Cartesian acceleration (both the linear and the angular) of the
	 /// end-effector during movements resulting from Cartesian-space commands (see Fig. 6). Note
	 /// that this command makes the robot come to a complete stop, even if blending is enabled.
	 /// Note that the argument OF THIS command is exceptionally limited TO 600. THIS is because
	 /// in firmware 8, a change was made to allow the robot to accelerate much faster. For backwards
	 /// compatibility, however, 100% now corresponds to 100% in firmware 7 and before.
	 /// Subindex 1 is the percentage of maximum Cartesian accelerations, ranging from 0.001 to 100.
	 SET_CART_ACC := 12,
	
	 /// This command defines the pose of the TRF with respect to the FRF. Note that this command
	 /// makes the robot come to a complete stop, even if blending is enabled.
	 /// Subindices 1, 2, 3 are in mm and 4, 5, 6 are in degrees. 
	 SET_TRF := 13,
	
	 /// This command defines the pose of the WRF with respect to the BRF. Note that this com-
	 /// mand makes the robot come to a complete stop, even if blending is enabled.
	 /// Subindices 1, 2, 3 are in mm and 4, 5, 6 are in degrees. 
	 SET_WRF := 14,
	
	 /// This command sets the desired robot inverse kinematic configuration to be observed in the
	 /// MovePose command.
	 /// The robot inverse kinematic configuration (see Fig. 5) can be automatically selected by
	 /// using the SetAutoConf command. Using SetConf automatically disables the automatic con-
	 /// figuration selection.
	 /// Subindices 1, 2, and 3 are -1 or 1.
	 SET_CONF := 15,
	
	 /// This command enables or disables the automatic robot configuration selection and has effect
	 /// only on the MovePose command. This automatic selection allows the controller to choose
	 /// the "closest" joint set corresponding to the desired pose (the arguments of the MovePose
	 /// command) and for which Euler Angle 6 is in the range +/-180° 
	 /// Subindex 1 is 0 or 1.
	 SET_AUTO_CONF := 16,
	
	 /// This command defines a checkpoint in the motion queue. Thus, if you send a sequence
	 /// of motion commands to the robot, then the command SetCheckpoint, then other motion
	 /// commands, you will be able to know the exact moment when the motion command sent just
	 /// before the SetCheckpoint command was completed. At that precise moment, the robot will
	 /// send you back the response [3030][n], where n is a positive integer number defined by you. If
	 /// blending was activated, the checkpoint response will be sent somewhere along the blending.
	 /// Finally, note that you can use the same checkpoint number multiple times.
	 /// Using a checkpoint is the only reliable way to know whether a particular motion sequence
	 /// was completed. Do not rely on the EOM or EOB messages as they may be received well
	 /// before the completion of a motion or a motion sequence (or, of course, not at all, if these
	 /// messages were not enabled).
	 /// Subindex 1 in an integer number, ranging from 1 to 8,000.
	 SET_CHECKPOINT := 17,
	
	 /// This command is used to open or close Mecademic's optional MEGP 25 gripper.
	 /// The gripper will move its fingers apart or closer until the grip force reaches 40 N. You can
	 /// reduce this maximum grip force with the SetGripperForce command. In addition, you can
	 /// control the speed of the gripper with the SetGripperVel command.
	 /// It is very important to understand that the GripperOpen and GripperClose commands
	 /// have the same behavior as a robot motion command, being executed only after the preceding
	 /// motion command has been completed. Currently, however, if a robot motion command is
	 /// sent after the GripperOpen or GripperClose command, the robot will start executing the
	 /// motion command without waiting for the gripper to finish its action. You must therefore
	 /// send a Delay command after GripperOpen and GripperClose commands.
	 /// Subindex 1 is 0 for GripperClose, and 1 for GripperOpen.
	 GRIPPER := 18,
	
	 /// This command limits the velocity of the gripper fingers (with respect to the gripper).
	 /// Subindex 1 is the percentage of maximum eger velocity (~100 mm/s), from 10 to 100.
	 SET_GRIPPER_VEL := 19,
	
	 /// This command limits the grip force of the MEGP 25 gripper.
	 /// Subindex 1 is the percentage of maximum grip force (~40 N), from 10 to 100.
	 SET_GRIPPER_FORCE := 20,
	
	 /// This command makes the robot rotate simultaneously its joints with the specified joint
	 /// velocities. All joint rotations start and stop at the same time. The path that the robot
	 /// takes is linear in the joint space, but nonlinear in the Cartesian space. Therefore, the TCP
	 /// path is not easily predictable (Fig. 7). With MoveJointsVel, the robot can cross singularities
	 /// without any problem.
	 /// Note that the robot will decelerate to a full stop after a period defined by the command
	 /// SetVelTimeout, unless another MoveJointsVel command is sent. Also, bear in mind that
	 /// the MoveJointsVel command, unlike position-mode motion commands, generates no motion
	 /// errors when a joint limit is reached. The robot simply stops slightly before the limit.
	 /// Subindices 1 trhough 6 are in °/s. 
	 MOVE_JOINTS_VEL := 21, 
	
	 /// This command makes the robot move its TRF with the specified instantaneous Cartesian
	 /// velocity, defined with respect to the WRF.
	 /// Note that the robot will decelerate to a complete stop after a period of time defined
	 /// by the SetVelTimeout command, unless another MoveLinVelWRF or a MoveLinVelTRF
	 /// command is sent and, of course, unless a PauseMotion command is sent or some motion
	 /// limit is encountered. Also, bear in mind that this command, unlike position-mode motion
	 /// commands, generates no motion errors when a joint limit (including the +/-180° limit on
	 /// joint 6) or a singularity is reached. The robot simply stops slightly before the limit.
	 /// Subindices 1, 2, 3 are in mm/s and 4, 5, 6 are in are in °/s.
	 MOVE_LIN_VEL_WRF := 22,
	
	 /// This command makes the robot move its TRF with the specified instantaneous Cartesian
	 /// velocity, defined with respect to the TRF.
	 /// Note that the robot will decelerate to a complete stop after a period of time defined
	 /// by the SetVelTimeout command, unless another MoveLinVelTRF or a MoveLinVelWRF
	 /// command is sent and, of course, unless a PauseMotion command is sent or some motion
	 /// limit is encountered. Also, bear in mind that this command, unlike position-mode motion
	 /// commands, generates no motion errors when a joint limit (including the +/-180° limit on
	 /// joint 6) or a singularity is reached. The robot simply stops slightly before the limit.
	 /// Subindices 1, 2, 3 are in mm/s and 4, 5, 6 are in are in °/s. 
	 MOVE_LIN_VEL_TRF := 23,
	  
	 /// This command sets the timeout after a velocity-mode motion command (MoveJointsVel,
	 /// MoveLinVelTRF, or MoveLinVelWRF), after which all joint speeds will be set to zero unless
	 /// another velocity-mode motion command is received. The SetVelTimeout command should
	 /// be regarded simply as a safety precaution.
	 /// Subindex 1 is in seconds.
	 SET_VEL_TIMEOUT := 24,
	  
	 /// THIS command sets the desired turn configuration FOR joint 6 TO be observed in the MovePose AND
	 /// MoveLin* commands (see Section 1.2.1 and Section 1.2.2). When a turn configuration is set, a MovePose
	 /// command is executed only if the final robot position can be in the desired turn configuration. In
	 /// contrast, when a desired turn configuration is set, a MoveLin* command will be executed only if the
	 /// final robot position can be and the initial robot position already is in the desired turn configuration. The
	 /// turn configuration can be automatically selected, when executing a MovePose or MoveLin* command,
	 /// by using the SetAutoConf command. Using SetConfTurn automatically disables the automatic turn
	 /// configuration selection.
	 /// Subindex 1  turn configuration, an integer between −100 AND 100.
	 /// The turn configuration parameter defines the desired range for joint 6, according to the following
	 /// equation: −180° + ct360° < θ6 ≤ 180° + ct360°).
	 SET_CONF_TURN	:= 25,
		
	 /// This command enables or disables the automatic turn selection for joint 6.
	 /// It affects the MovePose command, and all MoveLin* commands. When the automatic turn
	 /// selection is enabled, and a MovePose command is executed, joint 6 will always take the shortest path,
	 /// and rotate no more than 180°. In the case of a MoveLin* command, however, enabling the automatic
	 /// turn selection simply allows the change of turn configuration along the linear move.
	 /// Subindex1 enable (1) or disable (0) automatic turn configuration selection.
	 SET_AUTO_CONF_TURN := 26,
		
	 /// THIS command sets the thresholds FOR the torques applied TO each joint, as percentages OF the maximum
	 /// allowable torques that can be applied at each joint. When a torque limit is exceeded, a customizable
	 /// event is created. The event behavior can be set by the command SetTorqueLimitsCfg.
	 /// This command is intended only for improving the chances of protecting your robot, its end-effector, and
	 /// the surrounded equipment, in the case of a collision. The torque in each joint is estimated by measuring
	 /// the current in the corresponding drive.
	 /// Unlike the SetJointLimits commands, the SetTorqueLimits command can only be applied after the
	 /// robot has been homed. Note that high accelerations or large movements may also produce high torque
	 /// peaks. Therefore, you should rely on this command only in the vicinity of obstacles, for example, while
	 /// applying an adhesive. Remember that SetTorqueLimits is a motion command and will therefore be
	 /// inserted in the motion queue and not necessarily executed immediately.
	 /// Subindex 1,2,3,4,5,6 percentage of the maximum allowable torque that can be applied at joint i,
	 /// ranging from 0.001% to 100%.
	 SET_TORQUE_LIMITS := 27,
		
	 /// THIS command sets the robot behavior when a joint torque exceeds the threshold set BY the
	 /// SetTorqueLimits command. It also sets the filtering TYPE used FOR accurate detection. It also sends a
	 /// torque limit status every time torque limit status changes (exceeded or not) for events severity greater
	 /// than 0. Torque limit error is sent when torque exceeds the limit for severity 4.
	 /// Arguments :
	 /// • s: integer defining the torque limit event severity as
	 /// – 0, no action;
	 /// – 1, trace warning;
	 /// – 2, pause motion;
	 /// – 3, clear motion;
	 /// – 4, error.
	 /// • m: integer defining the detection mode as 0, always detect; 1, skip detection during acceleration/
	 /// deceleration and blending.
	 SET_TORQUE_LIMIT_CFG := 28,
		  
	 /// THIS command has the exact behavior as the MoveJoints command, but instead OF accepting the
	 /// desired (target) joint set as arguments, it takes the desired relative joint displacements. The command is
	 /// particularly useful when you need to displace certain joints a certain amount, but you do not know the
	 /// current joint position and wish to avoid having to use the command GetRtTargetJointPos.
	 /// Arguments :
	 /// • Δθi: the desired relative displacement of joint i (i = 1, 2, ..., 6), in degrees. The value of the argument
	 /// can be positive, negative or even zero.  
	 MOVE_JOINTS_REL := 29,
		  
	 /// THIS command is use TO control independently each OF the two valves in the MPM500 pneumatic module.
	 /// Arguments
	 /// • v1: open (1), close (0) or keep unchanged (−1) valve 1;
	 /// • v2: open (1), close (0) or keep unchanged (−1) valve 2.  
	 SET_VALVE_STATE := 30,
		
	 /// THIS command sets the closed AND open states OF the gripper AND is used mainly TO redefine the actions
	 /// of the GripperClose and GripperOpen commands, respectively. The SetGripperRange command is
	 /// useful for the MEGP 25LS gripper. If, for example, you are manipulating parts that require fingers
	 /// opening between 10 mm and 20 mm, but the allowable range of the gripper as detected during
	 /// the homing is 48 mm, it would be more efficient to redefine the actions of the GripperClose and
	 /// GripperOpen commands by calling SetGripperRange(8,22), or else the fingers will move more than
	 /// necessary, and therefore increase your cycle time.
	 /// The SetGripperRange command does not limit the accessible range of the gripper, in contrast to the
	 /// SetJointLimits command, which limits the range of a joint. For example, if during homing, the robot
	 /// detected that the range for the finger opening was [0, 15], and then you sent SetGripperRange(8,13),
	 /// you can still open the gripper more with MoveGripper(14). However, using the commands GripperOpen
	 /// and GripperClose will be equivalent to using the commands MoveGripper(8) and MoveGripper(13),
	 /// respectively. Furthermore, when the fingers opening is 8 mm (or less) or 13 mm (or more), the state of
	 /// the gripper will be “gripper open” or “gripper close”, respectively (see GetRtGripperState).
	 /// Arguments
	 /// • dclosed: fingers opening that should correspond to closed state, in mm;
	 /// • dopen: fingers opening that should correspond to open state, in mm.  
	 SET_GRIPPER_RANGE := 31,
		
	 /// The MEGP 25E AND MEGP 25LS grippers are equipped with incremental encoders, so it is impossible TO
	 /// directly measure the absolute positions of the gripper jaws. Thus, during the homing of the robot, the
	 /// gripper is also homed by completely closing and then opening its fingers, until resistance is met in each
	 /// direction. The maximum fingers opening is detected and is a positive number not larger than 6 mm
	 /// (MEGP 25E) or 48 mm (MEGP 25LS). Most importantly, the fingers opening, a non-negative distance,
	 /// is defined as the sum of the distances traveled by each jaw from their fully-closed positions detected
	 /// during homing.
	 /// The MoveGripper command makes the gripper fingers move towards the specified fingers opening.
	 /// Arguments :
	 /// • d: desired fingers opening, a  
	 MOVE_GRIPPER := 32,
		  
	 ///In revision 4 OF the Meca500, we have introduced the possibility TO go beyond the maximum rated joint
	 ///velocities in any type of movement. For compatibility reasons, we introduced this new command.
	 ///TheSetJointVelLimit overrides the default joint velocity limits. Unlike the SetJointVel command, this
	 ///command affects the movements generated by all Move* commands (even the MoveLinVel* ones).
	 ///Arguments :
	 ///• po: percentage of top rated joint velocities, ranging from 0.001 to 100, for R3, and to 150, for R4.
	 ///Default values
	 ///By default, po = 100.
	 ///As already mentioned in the SetJointVel command, in both revisions of Meca500, the top rated velocity
	 ///of joints 1 and 2 is 150°/s, of joint 3 is 180°/s, of joints 4 and 5 is 300°/s, and of joint 6 is 500°/s. 
	 ///In the case of the R4, the maximum velocity of each joint can be increased up to 225°/s 
	 ///for joints 1, 2 and 3,and up to 350°/s for joints 4 and 5. 
	 ///The velocity of joint 6 cannot be increased over its top rated limit of 500°/s. 
	 ///Thus, for example, if po = 140, the velocity of joints 1 and 2 will be limited to min(150*1.4, 225) = 210°/s, 
	 ///the velocity of joint 3 will be limited to min(180*1.4, 225) = 225°/s, etc., during a MoveLin motion.
	 SET_JOINT_VEL_LIMIT:=33, 
		  
	 /// THIS command starts a PROGRAM that has been previously saved in the robot's memory. The robot must
	 /// be activated and homed before running a program. Executing this command will launch the program n
	 /// only once.
	 /// Alternately, pressing the Start/Stop button on the robot base will start program 1 (and only program 1)
	 /// and execute it the number of times defined by the SetOfflineProgramLoop command.
	 /// Arguments
	 /// • n: program number, where n ≤ 500 (maximum number of programs that can be stored).  
	 START_PROGRAM := 100
)UINT;
END_TYPE

// Device/Application/F1000_UDTs/UDT_Meca500/STRUCT/Meca500
TYPE Meca500 :
STRUCT
Inputs : Meca500_Inputs;
Outputs : Meca500_Outputs;
	
END_STRUCT
END_TYPE

// Device/Application/F1000_UDTs/UDT_Meca500/STRUCT/Meca500_Inputs/Meca500_DynamicData
TYPE Meca500_DynamicData :
STRUCT
	DynamicDataTypeID	:	UDINT;	//Dynamic data type
	DynamicDataValue	:	ARRAY[0..5] OF REAL;	//Associated value
	
END_STRUCT
END_TYPE

// Device/Application/F1000_UDTs/UDT_Meca500/STRUCT/Meca500_Inputs/Meca500_Inputs
TYPE Meca500_Inputs :
STRUCT
	Status :	Meca500_Status;
	Motion	:	Meca500_Motion;
	Joint_set		:	ARRAY[0..5] OF REAL;
	EndEffetor_Pose	:	ARRAY[0..5] OF REAL;
	Configurations	:	ARRAY[0..3] OF SINT;
	WRF				:	ARRAY[0..5] OF REAL;
	TRF				:	ARRAY[0..5] OF REAL;
	TimeStamp	:	Meca500_TimeStamp;
	Reserved1	:	DINT;
	Reserved2	:	DINT;
	Reserved3	:	DINT;
	DynamicData	:	ARRAY[0..3] OF Meca500_DynamicData;
END_STRUCT
END_TYPE

// Device/Application/F1000_UDTs/UDT_Meca500/STRUCT/Meca500_Inputs/Meca500_Motion
TYPE Meca500_Motion :
STRUCT
	CheckPoint			:	UDINT;	//Indicates the last checkpoint number reached.
	MoveID				:	UINT;	//Acknowledges the MoveID of the last motion command queued for execution.
	FifoSpace			:	UINT;	//The number of commands that can be added to the robot's motion queue.
	MotionStatus		:	Meca500_MotionStatus;
	OfflineProgramID	:	UINT;	//ID of the offline program currently running (0 if none).
	
END_STRUCT
END_TYPE

// Device/Application/F1000_UDTs/UDT_Meca500/STRUCT/Meca500_Inputs/Meca500_MotionStatus
TYPE Meca500_MotionStatus :
STRUCT
	Paused				:	BIT;	//Indicates whether the motion is paused.
	EOB					:	BIT;
	EOM					:	BIT;
	FifoCleared			:	BIT;	//Indicates whether the motion queue is cleared.
	Pstop2				:	BIT;	//Indicates whether the P-Stop 2 is set.
	ExcessiveTorque		:	BIT;	//Indicates whether a joint torque is exceeding the user-defined torque limit.
	PStop2Resettable	:	BIT;	//ndicates whether the P-Stop 2 is removed, but is not reset yet.
	Reserved8			:	BIT;
	Reserved9			:	BIT;
	Reserved10			:	BIT;
	Reserved11			:	BIT;
	Reserved12			:	BIT;
	Reserved13			:	BIT;
	Reserved14			:	BIT;
	Reserved15			:	BIT;
	
END_STRUCT
END_TYPE

// Device/Application/F1000_UDTs/UDT_Meca500/STRUCT/Meca500_Inputs/Meca500_RobotStatus
TYPE Meca500_RobotStatus :
STRUCT 
	Busy 			: 	BIT;	//True only while the robot is being activated, homed or deactivated.
	Activated 		:	BIT;	//Indicates whether the motors are on (powered).
	Homed			:	BIT;	//Indicates whether the robot is homed and ready to receive motion commands.
	SimActivated	:	BIT;	//Indicates whether the robot simulation mode is activated.
	BrakesEngaged	:	BIT;	//Indicates whether the brakes are engaged.
	Recoverymode	:	BIT;	//Indicates whether the robot recovery mode is activated.
	EStop			:	BIT;	//Indicates whether the E-Stop is activated (Meca500 R4 only).
	Reserved7		:	BIT;
	Reserved8		:	BIT;
	Reserved9		:	BIT;
	Reserved10		:	BIT;
	Reserved11		:	BIT;
	Reserved12		:	BIT;
	Reserved13		:	BIT;
	Reserved14		:	BIT;
	Reserved15		:	BIT;

END_STRUCT
END_TYPE

// Device/Application/F1000_UDTs/UDT_Meca500/STRUCT/Meca500_Inputs/Meca500_Status
TYPE Meca500_Status :
STRUCT
	RobotStatus	:	Meca500_RobotStatus;
	ErrorCode		:	UINT;	//Indicates the error code or 0, if there is no error.
END_STRUCT	
END_TYPE

// Device/Application/F1000_UDTs/UDT_Meca500/STRUCT/Meca500_Inputs/Meca500_TimeStamp
TYPE Meca500_TimeStamp :
STRUCT
	Seconds				:	UDINT;	//Robot's monotonic timestamp (seconds) based on arbitrary reference.
	MicroSeconds		:	UDINT;	//Robot's monotonic timestamp (microseconds within second)
	DynamicDataCycles	:	UDINT;	//Number of times all available dynamic data has been refreshed
END_STRUCT
END_TYPE

// Device/Application/F1000_UDTs/UDT_Meca500/STRUCT/Meca500_Outputs/Meca500_BrakeControl
TYPE Meca500_BrakeControl :
STRUCT
	BrakesControlAllowed	:	BIT;	//Must be set to True to allow brakes control through cyclic data.
	BrakesEngaged			:	BIT;	//if set to True the brakes are engaged, ignored if the robot is activated.
	Reserved2			:	BIT;
	Reserved3			:	BIT;
	Reserved4			:	BIT;
	Reserved5			:	BIT;
	Reserved6			:	BIT;
	Reserved7			:	BIT;
	Reserved8			:	BIT;
	Reserved9			:	BIT;
	Reserved10			:	BIT;
	Reserved11			:	BIT;
	Reserved12			:	BIT;
	Reserved13			:	BIT;
	Reserved14			:	BIT;
	Reserved15			:	BIT;
	Reserved16			:	BIT;
	Reserved17			:	BIT;
	Reserved18			:	BIT;
	Reserved19			:	BIT;
	Reserved20			:	BIT;
	Reserved21			:	BIT;
	Reserved22			:	BIT;
	Reserved23			:	BIT;
	Reserved24			:	BIT;
	Reserved25			:	BIT;
	Reserved26			:	BIT;
	Reserved27			:	BIT;
	Reserved28			:	BIT;
	Reserved29			:	BIT;
	Reserved30			:	BIT;
	Reserved31			:	BIT;
END_STRUCT
END_TYPE

// Device/Application/F1000_UDTs/UDT_Meca500/STRUCT/Meca500_Outputs/Meca500_MotionCommand
TYPE Meca500_MotionCommand :
STRUCT
	MoveCommand	:	UDINT;
	Argument0	:	REAL;
	Argument1	:	REAL;
	Argument2	:	REAL;
	Argument3	:	REAL;
	Argument4	:	REAL;
	Argument5	:	REAL;
END_STRUCT
END_TYPE

// Device/Application/F1000_UDTs/UDT_Meca500/STRUCT/Meca500_Outputs/Meca500_MotionControl
TYPE Meca500_MotionControl :
STRUCT
	SetPoint	:	BIT;	//Has to be set to True for motion commands to be sent to the robot.
	PauseMotion	:	BIT;	//Puts the robot in pause without clearing the commands in the queue.
	ClearMotion	:	BIT;	//Clears the motion queue and puts the robot in pause.
	ResetPStop2	:	BIT;	//Resets P-Stop 2.
(*	Reserved4			:	BIT;
	Reserved5			:	BIT;
	Reserved6			:	BIT;
	Reserved7			:	BIT;
	Reserved8			:	BIT;
	Reserved9			:	BIT;
	Reserved10			:	BIT;
	Reserved11			:	BIT;
	Reserved12			:	BIT;
	Reserved13			:	BIT;
	Reserved14			:	BIT;
	Reserved15			:	BIT;
	*)
END_STRUCT
END_TYPE

// Device/Application/F1000_UDTs/UDT_Meca500/STRUCT/Meca500_Outputs/Meca500_Outputs
TYPE Meca500_Outputs :
STRUCT
	RobotControl	:	Meca500_RobotControl;
	MoveID		:	UINT;	//the change of which triggers the addition of the command specified in MotionCommandID to the motion queue.
	MotionControl	:	Meca500_MotionControl;
	MotionCommand	:	Meca500_MotionCommand;
	HostTime				:	UDINT;	//Current time in seconds since epoch.If non-zero, the robot will update its own time to this value
	BrakeControl			:	Meca500_BrakeControl;
	DynamicDataCfg0			:	UDINT;	//Dynamic data type for DynamicData[0]
	DynamicDataCfg1			:	UDINT;	//Dynamic data type for DynamicData[1]
	DynamicDataCfg2			:	UDINT;	//Dynamic data type for DynamicData[2]
	DynamicDataCfg3			:	UDINT;	//Dynamic data type for DynamicData[3]
END_STRUCT
END_TYPE

// Device/Application/F1000_UDTs/UDT_Meca500/STRUCT/Meca500_Outputs/Meca500_RobotControl
TYPE Meca500_RobotControl :
STRUCT
	Deactivate			:	BIT;	//Deactivates the robot when set to True.	
	Activate			:	BIT;	//Activates the robot when set to True(only if Deactivate bit is False).
	Home				:	BIT;	//Homes the robot when set to True (if activated but not homed).
	ResetError			:	BIT;	//Resets the error when set to True.
	EnableSimulation	:	BIT;	//Enables(True) OR disables(False) the simulation mode (only applied when the robot is deactivated).
	EnableRecoverymode	:	BIT;	//Enables(True) or disables(False) the recovery mode.
	Reserved6			:	BIT;
	Reserved7			:	BIT;
	Reserved8			:	BIT;
	Reserved9			:	BIT;
	Reserved10			:	BIT;
	Reserved11			:	BIT;
	Reserved12			:	BIT;
	Reserved13			:	BIT;
	Reserved14			:	BIT;
	Reserved15			:	BIT;
	Reserved16			:	BIT;
	Reserved17			:	BIT;
	Reserved18			:	BIT;
	Reserved19			:	BIT;
	Reserved20			:	BIT;
	Reserved21			:	BIT;
	Reserved22			:	BIT;
	Reserved23			:	BIT;
	Reserved24			:	BIT;
	Reserved25			:	BIT;
	Reserved26			:	BIT;
	Reserved27			:	BIT;
	Reserved28			:	BIT;
	Reserved29			:	BIT;
	Reserved30			:	BIT;
	Reserved31			:	BIT;
	
END_STRUCT
END_TYPE

// Device/Application/F100_VARs/GVL
{attribute 'qualified_only'}
VAR_GLOBAL
		Meca500_1 : Meca500;
		CAM_1: UDT_VS_Series;
		SYS: UDT_SYS;
		PARTX: UDT_PARTX;
		SF:SAFEBOOL;
END_VAR

// Device/Application/F001_ROBOT/F001_SR00_MAIN
PROGRAM F001_SR00_MAIN
VAR
END_VAR

(* body of a kind this reader does not render *)

END_PROGRAM

// Device/Application/F002_PART_X/F002_SR00_MAIN
PROGRAM F002_SR00_MAIN
VAR
END_VAR

(* body of a kind this reader does not render *)

END_PROGRAM

// Device/Application/PLC_PRG
PROGRAM PLC_PRG
VAR
	//Demo without function block control
	SequenceStep:INT;
	StartSequence:BOOL;
	
	//demo with function block control 
	TestSquareMove:BOOL;
	StepSquareMove:INT;
	LastStep:INT;
	Sent:BOOL;
	Buffered:BOOL;
	Error:BOOL;
	
	//Function Block instances
	MoveJoints:MoveJoints;
	SetCheckpoint:SetCheckpoint;
	MovePose:Movepose;
	Movelin:MoveLinRelTrf;
	SetCartLinVel:SetCartLinVel;
	
	//Positions for sequence
	ZeroJointsValues:ARRAY[0..5]OF REAL := [0,0,0,0,0,0];
	MovePoseValues:ARRAY[0..5]OF REAL := [100, 0, 200, 0, 180, 0];
	MoveLinValues1:ARRAY[0..5]OF REAL := [50, 0, 0, 0, 0, 0];
	MoveLinValues2:ARRAY[0..5]OF REAL := [0, 50, 0, 0, 0, 0];
	MoveLinValues3:ARRAY[0..5]OF REAL := [-50 ,0, 0, 0, 0, 0];
	MoveLinValues4:ARRAY[0..5]OF REAL := [0 ,-50, 0, 0, 0, 0];
//	CalculateWRF1: CalculateWRF;
	result: array[0..5] of real;
	point1: array[0..2] of real := [50,25,0];
	point2: array[0..2] of real := [175,25,10];
	point3: array[0..2] of real := [150,35,25];
END_VAR





//**********************************************************************************************************//
//Demo program using only the robot outputs
//Activate StartSequence to Start Demo
IF GVL.Meca500_1.Inputs.Status.RobotStatus.Activated AND GVL.Meca500_1.Inputs.Status.RobotStatus.Homed THEN
	IF StartSequence THEN
		GVL.Meca500_1.Outputs.MoveID:=1;
		SequenceStep := 10;
	END_IF		
	
	CASE SequenceStep OF
			//MoveJoints(0,0,0,0,0,0)
		10:	GVL.Meca500_1.Outputs.MotionControl.SetPoint:=TRUE;
			GVL.Meca500_1.Outputs.MotionCommand.MoveCommand:=1;
			GVL.Meca500_1.Outputs.MotionCommand.Argument0:=0;
			GVL.Meca500_1.Outputs.MotionCommand.Argument1:=0;
			GVL.Meca500_1.Outputs.MotionCommand.Argument2:=0;
			GVL.Meca500_1.Outputs.MotionCommand.Argument3:=0;
			GVL.Meca500_1.Outputs.MotionCommand.Argument4:=0;
			GVL.Meca500_1.Outputs.MotionCommand.Argument5:=0;
			GVL.Meca500_1.Outputs.MoveID:=10;
			StartSequence:=FALSE;	
			SequenceStep:=20;
			
			//MovePose(170,50,150,0,90,0)
		20:	GVL.Meca500_1.Outputs.MotionCommand.MoveCommand:=2;
			GVL.Meca500_1.Outputs.MotionCommand.Argument0:=170;
			GVL.Meca500_1.Outputs.MotionCommand.Argument1:=50;
			GVL.Meca500_1.Outputs.MotionCommand.Argument2:=150;
			GVL.Meca500_1.Outputs.MotionCommand.Argument3:=0;
			GVL.Meca500_1.Outputs.MotionCommand.Argument4:=90;
			GVL.Meca500_1.Outputs.MotionCommand.Argument5:=0;
			GVL.Meca500_1.Outputs.MoveID:=20;
			SequenceStep:=30;
			
			//MoveLin(170,-50,150,0,90,0)
		30:	GVL.Meca500_1.Outputs.MotionCommand.MoveCommand:=3;
			GVL.Meca500_1.Outputs.MotionCommand.Argument0:=170;
			GVL.Meca500_1.Outputs.MotionCommand.Argument1:=-50;
			GVL.Meca500_1.Outputs.MotionCommand.Argument2:=150;
			GVL.Meca500_1.Outputs.MotionCommand.Argument3:=0;
			GVL.Meca500_1.Outputs.MotionCommand.Argument4:=90;
			GVL.Meca500_1.Outputs.MotionCommand.Argument5:=0;
			GVL.Meca500_1.Outputs.MoveID:=30;
			SequenceStep:=40;
			
			//MoveLin(270,-50,150,0,90,0)
		40:	GVL.Meca500_1.Outputs.MotionCommand.MoveCommand:=3;
			GVL.Meca500_1.Outputs.MotionCommand.Argument0:=270;
			GVL.Meca500_1.Outputs.MotionCommand.Argument1:=-50;
			GVL.Meca500_1.Outputs.MotionCommand.Argument2:=150;
			GVL.Meca500_1.Outputs.MotionCommand.Argument3:=0;
			GVL.Meca500_1.Outputs.MotionCommand.Argument4:=90;
			GVL.Meca500_1.Outputs.MotionCommand.Argument5:=0;
			GVL.Meca500_1.Outputs.MoveID:=40;
			SequenceStep:=50;
			
			//MoveLin(270,50,150,0,90,0)
		50:	GVL.Meca500_1.Outputs.MotionCommand.MoveCommand:=3;
			GVL.Meca500_1.Outputs.MotionCommand.Argument0:=270;
			GVL.Meca500_1.Outputs.MotionCommand.Argument1:=50;
			GVL.Meca500_1.Outputs.MotionCommand.Argument2:=150;
			GVL.Meca500_1.Outputs.MotionCommand.Argument3:=0;
			GVL.Meca500_1.Outputs.MotionCommand.Argument4:=90;
			GVL.Meca500_1.Outputs.MotionCommand.Argument5:=0;
			GVL.Meca500_1.Outputs.MoveID:=50;
			SequenceStep:=60;
		
			//MoveLin(170,50,150,0,90,0)
		60:	GVL.Meca500_1.Outputs.MotionCommand.MoveCommand:=3;
			GVL.Meca500_1.Outputs.MotionCommand.Argument0:=170;
			GVL.Meca500_1.Outputs.MotionCommand.Argument1:=50;
			GVL.Meca500_1.Outputs.MotionCommand.Argument2:=150;
			GVL.Meca500_1.Outputs.MotionCommand.Argument3:=0;
			GVL.Meca500_1.Outputs.MotionCommand.Argument4:=90;
			GVL.Meca500_1.Outputs.MotionCommand.Argument5:=0;
			GVL.Meca500_1.Outputs.MoveID:=60;
			SequenceStep:=70;
			
			//MoveJoints(0,0,0,0,0,0)
		70:	GVL.Meca500_1.Outputs.MotionCommand.MoveCommand:=1;
			GVL.Meca500_1.Outputs.MotionCommand.Argument0:=0;
			GVL.Meca500_1.Outputs.MotionCommand.Argument1:=0;
			GVL.Meca500_1.Outputs.MotionCommand.Argument2:=0;
			GVL.Meca500_1.Outputs.MotionCommand.Argument3:=0;
			GVL.Meca500_1.Outputs.MotionCommand.Argument4:=0;
			GVL.Meca500_1.Outputs.MotionCommand.Argument5:=0;
			GVL.Meca500_1.Outputs.MoveID:=70;	
			SequenceStep:=80;
			
		80:GVL.Meca500_1.Outputs.MotionControl.SetPoint:=FALSE;
			SequenceStep:=0;	
			
			
	END_CASE	

END_IF	

//******************************************************************************************************************//
//Demo program using intructions
//Activate TestSquareMove to Start Demo
IF TestSquareMove THEN
	//Activate the robot if not activated
	GVL.Meca500_1.Outputs.RobotControl.Deactivate := false;
	IF GVL.Meca500_1.Inputs.Status.RobotStatus.Activated THEN 
		GVL.Meca500_1.Outputs.RobotControl.Activate := FALSE;
	ELSE	
		GVL.Meca500_1.Outputs.RobotControl.Activate := TRUE;	
	END_IF
	
	//Home the robot if not home
	IF GVL.Meca500_1.Inputs.Status.RobotStatus.Homed THEN
		GVL.Meca500_1.Outputs.RobotControl.Home:=FALSE;
	ELSE
		GVL.Meca500_1.Outputs.RobotControl.Home:=TRUE;
	END_IF

	IF	GVL.Meca500_1.Inputs.Status.RobotStatus.Activated AND GVL.Meca500_1.Inputs.Status.RobotStatus.Homed THEN
			CASE StepSquareMove OF
			0:	StepSquareMove:=1; //Unused Step
			SetCartLinVel(
				Velocity_limit:=10,
				Robot:=GVL.Meca500_1,
				Sent:=Sent,
				Error=>Error,
				Buffered:=Buffered
				);
			1:	StepSquareMove:=2; //Unused Step
			2:	MoveJoints(
					Joint_Angle:= ZeroJointsValues, 
					ExternalStatecontrol:=0 , 
					ExternalMoveID:=0 , 
					Robot:= GVL.Meca500_1 , 
					Error=> Error, 
					Sent:= Sent, 
					Buffered:= Buffered);
				
			3:	SetCheckpoint(
					CheckpointID:=3, 
					ExternalStatecontrol:=0 , 
					ExternalMoveID:=0 , 
					Robot:= GVL.Meca500_1 , 
					Error=> Error, 
					Sent:= Sent, 
					Buffered:= Buffered);	
			4:		IF gvl.Meca500_1.Inputs.Motion.CheckPoint=720899 THEN
					StepSquareMove:=5;
				END_IF	
				//StepSquareMove:=5;
				
			5:	MovePose(
					Pose:= MovePoseValues, 
					ExternalStatecontrol:=0 , 
					ExternalMoveID:=0 , 
					Robot:= 0 , 
					Error=> Error, 
					Sent:= Sent, 
					Buffered:= Buffered); 
			6:	MoveLin(
					Pose:= MoveLinValues1, 
					ExternalStatecontrol:=0 , 
					ExternalMoveID:=0 , 
					Robot:= GVL.Meca500_1 , 
					Error=> Error, 
					Sent:= Sent, 
					Buffered:= Buffered);
			7:	MoveLin(
					Pose:= MoveLinValues2, 
					ExternalStatecontrol:=0 , 
					ExternalMoveID:=0 , 
					Robot:= GVL.Meca500_1 , 
					Error=> Error, 
					Sent:= Sent, 
					Buffered:= Buffered);
			8:	MoveLin(
					Pose:= MoveLinValues3, 
					ExternalStatecontrol:=0 , 
					ExternalMoveID:=0 , 
					Robot:= GVL.Meca500_1 , 
					Error=> Error, 
					Sent:= Sent, 
					Buffered:= Buffered);
			9:	MoveLin(
					Pose:= MoveLinValues4, 
					ExternalStatecontrol:=0 , 
					ExternalMoveID:=0 , 
					Robot:= GVL.Meca500_1 , 
					Error=> Error, 
					Sent:= Sent, 
					Buffered:= Buffered);
			10:	MoveJoints(
					Joint_Angle:= ZeroJointsValues, 
					ExternalStatecontrol:=0 , 
					ExternalMoveID:=0 , 
					Robot:= GVL.Meca500_1 , 
					Error=> Error, 
					Sent:= Sent, 
					Buffered:= Buffered);
			11:	SetCheckpoint(
					CheckpointID:=11, 
					ExternalStatecontrol:=0 , 
					ExternalMoveID:=0 , 
					Robot:= GVL.Meca500_1 , 
					Error=> Error, 
					Sent:= Sent, 
					Buffered:= Buffered);	
			12:	IF gvl.Meca500_1.Inputs.Motion.CheckPoint=720907 THEN
					StepSquareMove:=13;
				END_IF
				//StepSquareMove:=13;
			13:	StepSquareMove:=0;			
			
			END_CASE
			
			//When command is sent and buffered, Reset those tag and go to next step
			IF Sent AND Buffered THEN
				StepSquareMove:=StepSquareMove+1;
				Sent:=0;
				Buffered:=0;
			END_IF 
			
		//If not Ready, return to Step 0	
		ELSE
			//Log when the robot stopped
			IF StepSquareMove > 0 THEN
				LastStep:=StepSquareMove;
			END_IF
			StepSquareMove:=0;
		END_IF		
Else
	StepSquareMove:=0;
	gvl.Meca500_1.Outputs.RobotControl.ResetError:=TRUE;
	IF GVL.Meca500_1.Inputs.Status.RobotStatus.Activated THEN 
		GVL.Meca500_1.Outputs.RobotControl.Activate := FALSE;
		GVL.Meca500_1.Outputs.RobotControl.Deactivate := true;
	end_if;
END_IF

END_PROGRAM

// Device/Application/F1000_FBs/Meca500/MoveJoints
FUNCTION_BLOCK MoveJoints
VAR_INPUT
	Joint_Angle				:	ARRAY[1..6]OF REAL;
	ExternalStatecontrol 	:	BOOL;
	ExternalMoveID			:	UINT;
END_VAR
VAR_IN_OUT
	Robot	:	Meca500;	
	Sent		:	BOOL;
	Buffered	:	BOOL;
END_VAR
VAR_OUTPUT
	Error		:	BOOL;

END_VAR
VAR
	Output_Params	:	ARRAY[1..6] OF REAL;
	FirstScan: BOOL;
END_VAR

        (*Collect Inputs and store them locally*)
Output_Params[1]:=Joint_Angle[1];
Output_Params[2]:=Joint_Angle[2];
Output_Params[3]:=Joint_Angle[3];
Output_Params[4]:=Joint_Angle[4];
Output_Params[5]:=Joint_Angle[5];
Output_Params[6]:=Joint_Angle[6];


(* If Values have change, Reinitialise Outputs*)

IF FirstScan=0 OR Robot.Outputs.MotionCommand.Argument0 <> Output_Params[1] OR Robot.Outputs.MotionCommand.Argument1 <> Output_Params[2] OR Robot.Outputs.MotionCommand.Argument2 <> Output_Params[3] OR Robot.Outputs.MotionCommand.Argument3 <> Output_Params[4] OR Robot.Outputs.MotionCommand.Argument4 <> Output_Params[5] OR Robot.Outputs.MotionCommand.Argument5 <> Output_Params[6] THEN
	Sent := FALSE;
	Buffered := FALSE;
END_IF;

(*if not in legacy mode, Act Setpoint*)
IF Robot.Outputs.MoveID <> 0 THEN
    Robot.Outputs.MotionControl.SetPoint := TRUE;
END_IF;

(* To send _Move, send _Move ID *)
IF NOT Buffered AND NOT Sent THEN
    
    Robot.Outputs.MotionCommand.MoveCommand := Meca500_MotionCommandID.MOVE_JOINTS ;
    Robot.Outputs.MotionCommand.Argument0 := Output_Params[1];
	Robot.Outputs.MotionCommand.Argument1 := Output_Params[2];
	Robot.Outputs.MotionCommand.Argument2 := Output_Params[3];
	Robot.Outputs.MotionCommand.Argument3 := Output_Params[4];
	Robot.Outputs.MotionCommand.Argument4 := Output_Params[5];
	Robot.Outputs.MotionCommand.Argument5 := Output_Params[6];
	
    
    IF ExternalStateControl THEN
        IF ExternalMoveID <> 0 AND ExternalMoveID <> 32010 AND ExternalMoveID <> 32011 THEN
            Robot.Outputs.MoveID := ExternalMoveID;
            Sent := TRUE;
        END_IF;
        
    ELSE (*Not External Control*)
        IF Robot.Outputs.MoveID = 32010 THEN
            Robot.Outputs.MoveID := 32011;
        ELSIF Robot.Outputs.MoveID = 32011 THEN
            Robot.Outputs.MoveID := 32010;
        ELSIF Robot.Outputs.MoveID <> 32010 OR Robot.Outputs.MoveID <> 32011 THEN
            Robot.Outputs.MoveID := 32010;
        END_IF;
        Sent := TRUE;
    END_IF;
END_IF;

(* Check if _Move has been sent, if so, check if it was received *)
IF Sent THEN
    IF Robot.Outputs.MotionCommand.MoveCommand = Meca500_MotionCommandID.MOVE_JOINTS THEN
        IF Robot.Outputs.MotionCommand.Argument0 = Output_Params[1] AND Robot.Outputs.MotionCommand.Argument1 = Output_Params[2] AND Robot.Outputs.MotionCommand.Argument2 = Output_Params[3] AND Robot.Outputs.MotionCommand.Argument3 = Output_Params[4] AND Robot.Outputs.MotionCommand.Argument4 = Output_Params[5] AND Robot.Outputs.MotionCommand.Argument5 = Output_Params[6] THEN
            IF Robot.Inputs.Motion.MoveID = Robot.Outputs.MoveID THEN
                Buffered := TRUE;
			//	Sent:=FALSE;
            END_IF;
        END_IF;
    END_IF;
END_IF;

(*If External _Move ID is equal to Internal, raise an error*)
IF ExternalMoveID = 32010 OR ExternalMoveID = 32011 THEN
    Error := TRUE;
END_IF;

FirstScan := TRUE;

END_FUNCTION_BLOCK

// Device/Application/F1000_FBs/Meca500/MovePose
FUNCTION_BLOCK MovePose
VAR_INPUT
	Pose					:	ARRAY[1..6]OF REAL;
	ExternalStatecontrol 	:	BOOL;
	ExternalMoveID			:	UINT;
END_VAR
VAR_IN_OUT
	Robot	:	Meca500;
	Sent		:	BOOL;
	Buffered	:	BOOL;	
END_VAR
VAR_OUTPUT
	Error		:	BOOL;

END_VAR
VAR
	Output_Params	:	ARRAY[1..6] OF REAL;
	i:INT;
	FirstScan	:	BOOL	:=0;
END_VAR

        (*Collect Inputs and store them locally*)
Output_Params[1]:=Pose[1];
Output_Params[2]:=Pose[2];
Output_Params[3]:=Pose[3];
Output_Params[4]:=Pose[4];
Output_Params[5]:=Pose[5];
Output_Params[6]:=Pose[6];


(* If Values have change, Reinitialise Outputs*)

IF FirstScan=0 OR Robot.Outputs.MotionCommand.Argument0 <> Output_Params[1] OR Robot.Outputs.MotionCommand.Argument1 <> Output_Params[2] OR Robot.Outputs.MotionCommand.Argument2 <> Output_Params[3] OR Robot.Outputs.MotionCommand.Argument3 <> Output_Params[4] OR Robot.Outputs.MotionCommand.Argument4 <> Output_Params[5] OR Robot.Outputs.MotionCommand.Argument5 <> Output_Params[6] THEN
	
	Sent := FALSE;
	Buffered := FALSE;

END_IF;


(*if not in legacy mode, Act Setpoint*)
IF Robot.Outputs.MoveID <> 0 THEN
    Robot.Outputs.MotionControl.SetPoint := TRUE;
END_IF;

(* To send _Move, send _Move ID *)
IF NOT Buffered AND NOT Sent THEN
    
    Robot.Outputs.MotionCommand.MoveCommand := Meca500_MotionCommandID.MOVE_POSE;
    Robot.Outputs.MotionCommand.Argument0 := Output_Params[1];
	Robot.Outputs.MotionCommand.Argument1 := Output_Params[2];
	Robot.Outputs.MotionCommand.Argument2 := Output_Params[3];
	Robot.Outputs.MotionCommand.Argument3 := Output_Params[4];
	Robot.Outputs.MotionCommand.Argument4 := Output_Params[5];
	Robot.Outputs.MotionCommand.Argument5 := Output_Params[6];
    
    IF ExternalStateControl THEN
        IF ExternalMoveID <> 0 AND ExternalMoveID <> 32020 AND ExternalMoveID <> 32021 THEN
            Robot.Outputs.MoveID := ExternalMoveID;
            Sent := TRUE;
        END_IF;
        
    ELSE (*Not External Control*)
        IF Robot.Outputs.MoveID = 32020 THEN
            Robot.Outputs.MoveID := 32021;
        ELSIF Robot.Outputs.MoveID = 32021 THEN
            Robot.Outputs.MoveID := 32020;
        ELSIF Robot.Outputs.MoveID <> 32020 OR Robot.Outputs.MoveID <> 32021 THEN
            Robot.Outputs.MoveID := 32020;
        END_IF;
        Sent := TRUE;
    END_IF;
END_IF;

(* Check if _Move has been sent, if so, check if it was received *)
IF Sent THEN
    IF Robot.Outputs.MotionCommand.MoveCommand = Meca500_MotionCommandID.MOVE_POSE THEN
        IF Robot.Outputs.MotionCommand.Argument0 = Output_Params[1] AND Robot.Outputs.MotionCommand.Argument1 = Output_Params[2] AND Robot.Outputs.MotionCommand.Argument2 = Output_Params[3] AND Robot.Outputs.MotionCommand.Argument3 = Output_Params[4] AND Robot.Outputs.MotionCommand.Argument4 = Output_Params[5] AND Robot.Outputs.MotionCommand.Argument5 = Output_Params[6] THEN
            IF Robot.Inputs.Motion.MoveID = Robot.Outputs.MoveID THEN
                Buffered := TRUE;
			//	Sent:=FALSE;
            END_IF;
        END_IF;
    END_IF;
END_IF;

(*If External _Move ID is equal to Internal, raise an error*)
IF ExternalMoveID = 32020 OR ExternalMoveID = 32021 THEN
    Error := TRUE;
END_IF;
FirstScan := TRUE;

END_FUNCTION_BLOCK

// Device/Application/F1000_FBs/Meca500/MoveLin
FUNCTION_BLOCK MoveLin
VAR_INPUT
	Pose					:	ARRAY[1..6]OF REAL;
	ExternalStatecontrol 	:	BOOL;
	ExternalMoveID			:	UINT;
END_VAR
VAR_IN_OUT
	Robot	:	Meca500;
	Sent		:	BOOL;
	Buffered	:	BOOL;
END_VAR
VAR_OUTPUT
	Error		:	BOOL;

END_VAR
VAR
	Output_Params	:	ARRAY[1..6] OF REAL;
	FirstScan: BOOL;
END_VAR

        (*Collect Inputs and store them locally*)
Output_Params[1]:=Pose[1];
Output_Params[2]:=Pose[2];
Output_Params[3]:=Pose[3];
Output_Params[4]:=Pose[4];
Output_Params[5]:=Pose[5];
Output_Params[6]:=Pose[6];


(* If Values have change, Reinitialise Outputs*)
IF FirstScan = 0 OR Robot.Outputs.MotionCommand.Argument0 <> Output_Params[1] OR Robot.Outputs.MotionCommand.Argument1 <> Output_Params[2] OR Robot.Outputs.MotionCommand.Argument2 <> Output_Params[3] OR Robot.Outputs.MotionCommand.Argument3 <> Output_Params[4] OR Robot.Outputs.MotionCommand.Argument4 <> Output_Params[5] OR Robot.Outputs.MotionCommand.Argument5 <> Output_Params[6] THEN
	Sent := FALSE;
	Buffered := FALSE;	

END_IF;

(*if not in legacy mode, Act Setpoint*)
IF Robot.Outputs.MoveID <> 0 THEN
    Robot.Outputs.MotionControl.SetPoint := TRUE;
END_IF;

(* To send _Move, send _Move ID *)
IF NOT Buffered AND NOT Sent THEN
    
    Robot.Outputs.MotionCommand.MoveCommand := Meca500_MotionCommandID.MOVE_LIN;
    Robot.Outputs.MotionCommand.Argument0 := Output_Params[1];
	Robot.Outputs.MotionCommand.Argument1 := Output_Params[2];
	Robot.Outputs.MotionCommand.Argument2 := Output_Params[3];
	Robot.Outputs.MotionCommand.Argument3 := Output_Params[4];
	Robot.Outputs.MotionCommand.Argument4 := Output_Params[5];
	Robot.Outputs.MotionCommand.Argument5 := Output_Params[6];
    
    IF ExternalStateControl THEN
        IF ExternalMoveID <> 0 AND ExternalMoveID <> 32030 AND ExternalMoveID <> 32031 THEN
            Robot.Outputs.MoveID := ExternalMoveID;
            Sent := TRUE;
        END_IF;
        
    ELSE (*Not External Control*)
        IF Robot.Outputs.MoveID = 32030 THEN
            Robot.Outputs.MoveID := 32031;
        ELSIF Robot.Outputs.MoveID = 32031 THEN
            Robot.Outputs.MoveID := 32030;
        ELSIF Robot.Outputs.MoveID <> 32030 OR Robot.Outputs.MoveID <> 32031 THEN
            Robot.Outputs.MoveID := 32030;
        END_IF;
        Sent := TRUE;
    END_IF;
END_IF;

(* Check if _Move has been sent, if so, check if it was received *)
IF Sent THEN
    IF Robot.Outputs.MotionCommand.MoveCommand = Meca500_MotionCommandID.MOVE_LIN THEN
        IF Robot.Outputs.MotionCommand.Argument0 = Output_Params[1] AND Robot.Outputs.MotionCommand.Argument1 = Output_Params[2] AND Robot.Outputs.MotionCommand.Argument2 = Output_Params[3] AND Robot.Outputs.MotionCommand.Argument3 = Output_Params[4] AND Robot.Outputs.MotionCommand.Argument4 = Output_Params[5] AND Robot.Outputs.MotionCommand.Argument5 = Output_Params[6] THEN
            IF Robot.Inputs.Motion.MoveID = Robot.Outputs.MoveID THEN
                Buffered := TRUE;
				//Sent:=FALSE;
            END_IF;
        END_IF;
    END_IF;
END_IF;

(*If External _Move ID is equal to Internal, raise an error*)
IF ExternalMoveID = 32030 OR ExternalMoveID = 32031 THEN
    Error := TRUE;
END_IF;
FirstScan := TRUE;

END_FUNCTION_BLOCK

// Device/Application/F1000_FBs/Meca500/SetCartLinVel
FUNCTION_BLOCK SetCartLinVel
VAR_INPUT
	Velocity_Limit					:	REAL;
	ExternalStatecontrol 	:	BOOL;
	ExternalMoveID			:	UINT;
END_VAR
VAR_IN_OUT
	Robot		:	Meca500;	
	Sent		:	BOOL;
	Buffered	:	BOOL;
END_VAR
VAR_OUTPUT
	Error		:	BOOL;
END_VAR
VAR
	Output_Params	:	ARRAY[1..6] OF REAL;
	FirstScan		:	BOOL;
END_VAR

        (*Collect Inputs and store them locally*)
Output_Params[1]:=Velocity_Limit;
Output_Params[2]:=0;
Output_Params[3]:=0;
Output_Params[4]:=0;
Output_Params[5]:=0;
Output_Params[6]:=0;


(* If Values have change, Reinitialise Outputs*)

IF FirstScan=0 OR Robot.Outputs.MotionCommand.Argument0 <> Output_Params[1] OR Robot.Outputs.MotionCommand.Argument1 <> Output_Params[2] OR Robot.Outputs.MotionCommand.Argument2 <> Output_Params[3] OR Robot.Outputs.MotionCommand.Argument3 <> Output_Params[4] OR Robot.Outputs.MotionCommand.Argument4 <> Output_Params[5] OR Robot.Outputs.MotionCommand.Argument5 <> Output_Params[6] THEN
	Buffered := FALSE;
	Sent := FALSE;
END_IF;

(*if not in legacy mode, Act Setpoint*)
IF Robot.Outputs.MoveID <> 0 THEN
    Robot.Outputs.MotionControl.SetPoint := TRUE;
END_IF;

(* To send _Move, send _Move ID *)
IF NOT Buffered AND NOT Sent THEN
    
    Robot.Outputs.MotionCommand.MoveCommand := Meca500_MotionCommandID.SET_CART_LIN_VEL;
    Robot.Outputs.MotionCommand.Argument0 := Output_Params[1];
	Robot.Outputs.MotionCommand.Argument1 := Output_Params[2];
	Robot.Outputs.MotionCommand.Argument2 := Output_Params[3];
	Robot.Outputs.MotionCommand.Argument3 := Output_Params[4];
	Robot.Outputs.MotionCommand.Argument4 := Output_Params[5];
	Robot.Outputs.MotionCommand.Argument5 := Output_Params[6];
    
    IF ExternalStateControl THEN
        IF ExternalMoveID <> 0 AND ExternalMoveID <> 32110 AND ExternalMoveID <> 32111 THEN
            Robot.Outputs.MoveID := ExternalMoveID;
            Sent := TRUE;
        END_IF;
        
    ELSE (*Not External Control*)
        IF Robot.Outputs.MoveID = 32110 THEN
            Robot.Outputs.MoveID := 32111;
        ELSIF Robot.Outputs.MoveID = 32111 THEN
            Robot.Outputs.MoveID := 32110;
        ELSIF Robot.Outputs.MoveID <> 32110 OR Robot.Outputs.MoveID <> 32111 THEN
            Robot.Outputs.MoveID := 32110;
        END_IF;
        Sent := TRUE;
    END_IF;
END_IF;

(* Check if _Move has been sent, if so, check if it was received *)
IF Sent THEN
    IF Robot.Outputs.MotionCommand.MoveCommand = Meca500_MotionCommandID.SET_CART_LIN_VEL THEN
        IF Robot.Outputs.MotionCommand.Argument0 = Output_Params[1] AND Robot.Outputs.MotionCommand.Argument1 = Output_Params[2] AND Robot.Outputs.MotionCommand.Argument2 = Output_Params[3] AND Robot.Outputs.MotionCommand.Argument3 = Output_Params[4] AND Robot.Outputs.MotionCommand.Argument4 = Output_Params[5] AND Robot.Outputs.MotionCommand.Argument5 = Output_Params[6] THEN
            IF Robot.Inputs.Motion.MoveID = Robot.Outputs.MoveID THEN
                Buffered := TRUE;
            END_IF;
        END_IF;
    END_IF;
END_IF;

(*If External _Move ID is equal to Internal, raise an error*)
IF ExternalMoveID = 32110 OR ExternalMoveID = 32111 THEN
    Error := TRUE;
END_IF;
FirstScan:=TRUE;

END_FUNCTION_BLOCK

// Device/Application/F1000_FBs/Meca500/SetCheckpoint
FUNCTION_BLOCK SetCheckpoint
VAR_INPUT
	CheckpointID					:	REAL;
	ExternalStatecontrol 	:	BOOL;
	ExternalMoveID			:	UINT;
END_VAR
VAR_IN_OUT
	Robot	:	Meca500;	
	Sent		:	BOOL;
	Buffered	:	BOOL;
END_VAR
VAR_OUTPUT
	Error		:	BOOL;
END_VAR
VAR
	Output_Params	:	ARRAY[1..6] OF REAL;
	i:INT;
	FirstScan: BOOL;
END_VAR

        (*Collect Inputs and store them locally*)
Output_Params[1]:=CheckpointID;
Output_Params[2]:=0;
Output_Params[3]:=0;
Output_Params[4]:=0;
Output_Params[5]:=0;
Output_Params[6]:=0;


(* If Values have change, Reinitialise Outputs*)

IF FirstScan=0 OR Robot.Outputs.MotionCommand.Argument0 <> Output_Params[1] OR Robot.Outputs.MotionCommand.Argument1 <> Output_Params[2] OR Robot.Outputs.MotionCommand.Argument2 <> Output_Params[3] OR Robot.Outputs.MotionCommand.Argument3 <> Output_Params[4] OR Robot.Outputs.MotionCommand.Argument4 <> Output_Params[5] OR Robot.Outputs.MotionCommand.Argument5 <> Output_Params[6] THEN
	Sent := FALSE;
	Buffered := FALSE;
END_IF;

(*if not in legacy mode, Act Setpoint*)
IF Robot.Outputs.MoveID <> 0 THEN
    Robot.Outputs.MotionControl.SetPoint := TRUE;
END_IF;

(* To send _Move, send _Move ID *)
IF NOT Buffered AND NOT Sent THEN
    
    Robot.Outputs.MotionCommand.MoveCommand := Meca500_MotionCommandID.SET_CHECKPOINT;
    Robot.Outputs.MotionCommand.Argument0 := Output_Params[1];
	Robot.Outputs.MotionCommand.Argument1 := Output_Params[2];
	Robot.Outputs.MotionCommand.Argument2 := Output_Params[3];
	Robot.Outputs.MotionCommand.Argument3 := Output_Params[4];
	Robot.Outputs.MotionCommand.Argument4 := Output_Params[5];
	Robot.Outputs.MotionCommand.Argument5 := Output_Params[6];
    
    IF ExternalStateControl THEN
        IF ExternalMoveID <> 0 AND ExternalMoveID <> 32170 AND ExternalMoveID <> 32171 THEN
            Robot.Outputs.MoveID := ExternalMoveID;
            Sent := TRUE;
        END_IF;
        
    ELSE (*Not External Control*)
        IF Robot.Outputs.MoveID = 32170 THEN
            Robot.Outputs.MoveID := 32171;
        ELSIF Robot.Outputs.MoveID = 32171 THEN
            Robot.Outputs.MoveID := 32170;
        ELSIF Robot.Outputs.MoveID <> 32170 OR Robot.Outputs.MoveID <> 32171 THEN
            Robot.Outputs.MoveID := 32170;
        END_IF;
        Sent := TRUE;
    END_IF;
END_IF;

(* Check if _Move has been sent, if so, check if it was received *)
IF Sent THEN
    IF Robot.Outputs.MotionCommand.MoveCommand = Meca500_MotionCommandID.SET_CHECKPOINT THEN
        IF Robot.Outputs.MotionCommand.Argument0 = Output_Params[1] AND Robot.Outputs.MotionCommand.Argument1 = Output_Params[2] AND Robot.Outputs.MotionCommand.Argument2 = Output_Params[3] AND Robot.Outputs.MotionCommand.Argument3 = Output_Params[4] AND Robot.Outputs.MotionCommand.Argument4 = Output_Params[5] AND Robot.Outputs.MotionCommand.Argument5 = Output_Params[6] THEN
            IF Robot.Inputs.Motion.MoveID = Robot.Outputs.MoveID THEN
                Buffered := TRUE;
			//	Sent:=FALSE;
            END_IF;
        END_IF;
    END_IF;
END_IF;

(*If External _Move ID is equal to Internal, raise an error*)
IF ExternalMoveID = 32170 OR ExternalMoveID = 32171 THEN
    Error := TRUE;
END_IF;
FirstScan := TRUE;

END_FUNCTION_BLOCK

// Device/Application/F1000_FBs/Meca500/MoveLinRelTrf
FUNCTION_BLOCK MoveLinRelTrf
VAR_INPUT
	Pose					:	ARRAY[1..6]OF REAL;
	ExternalStatecontrol 	:	BOOL;
	ExternalMoveID			:	UINT;
END_VAR
VAR_IN_OUT
	Robot	:	Meca500;	
	Sent		:	BOOL;
	Buffered	:	BOOL;
END_VAR
VAR_OUTPUT
	Error		:	BOOL;
END_VAR
VAR
	Output_Params	:	ARRAY[1..6] OF REAL;
	FirstScan: BOOL;
END_VAR

        (*Collect Inputs and store them locally*)
Output_Params[1]:=Pose[1];
Output_Params[2]:=Pose[2];
Output_Params[3]:=Pose[3];
Output_Params[4]:=Pose[4];
Output_Params[5]:=Pose[5];
Output_Params[6]:=Pose[6];


(* If Values have change, Reinitialise Outputs*)

    IF FirstScan=0 OR Robot.Outputs.MotionCommand.Argument0 <> Output_Params[1] OR Robot.Outputs.MotionCommand.Argument1 <> Output_Params[2] OR Robot.Outputs.MotionCommand.Argument2 <> Output_Params[3] OR Robot.Outputs.MotionCommand.Argument3 <> Output_Params[4] OR Robot.Outputs.MotionCommand.Argument4 <> Output_Params[5] OR Robot.Outputs.MotionCommand.Argument5 <> Output_Params[6] THEN
		Buffered := FALSE;
		Sent := FALSE;
	END_IF;

(*if not in legacy mode, Act Setpoint*)
IF Robot.Outputs.MoveID <> 0 THEN
    Robot.Outputs.MotionControl.SetPoint := TRUE;
END_IF;

(* To send _Move, send _Move ID *)
IF NOT Buffered AND NOT Sent THEN
    
    Robot.Outputs.MotionCommand.MoveCommand := Meca500_MotionCommandID.MOVE_LIN_REL_TRF;
    Robot.Outputs.MotionCommand.Argument0 := Output_Params[1];
	Robot.Outputs.MotionCommand.Argument1 := Output_Params[2];
	Robot.Outputs.MotionCommand.Argument2 := Output_Params[3];
	Robot.Outputs.MotionCommand.Argument3 := Output_Params[4];
	Robot.Outputs.MotionCommand.Argument4 := Output_Params[5];
	Robot.Outputs.MotionCommand.Argument5 := Output_Params[6];
    
    IF ExternalStateControl THEN
        IF ExternalMoveID <> 0 AND ExternalMoveID <> 32040 AND ExternalMoveID <> 32041 THEN
            Robot.Outputs.MoveID := ExternalMoveID;
            Sent := TRUE;
        END_IF;
        
    ELSE (*Not External Control*)
        IF Robot.Outputs.MoveID = 32040 THEN
            Robot.Outputs.MoveID := 32041;
        ELSIF Robot.Outputs.MoveID = 32041 THEN
            Robot.Outputs.MoveID := 32040;
        ELSIF Robot.Outputs.MoveID <> 32040 OR Robot.Outputs.MoveID <> 32041 THEN
            Robot.Outputs.MoveID := 32040;
        END_IF;
        Sent := TRUE;
    END_IF;
END_IF;

(* Check if _Move has been sent, if so, check if it was received *)
IF Sent THEN
    IF Robot.Outputs.MotionCommand.MoveCommand = Meca500_MotionCommandID.Move_LIN_REL_TRF THEN
        IF Robot.Outputs.MotionCommand.Argument0 = Output_Params[1] AND Robot.Outputs.MotionCommand.Argument1 = Output_Params[2] AND Robot.Outputs.MotionCommand.Argument2 = Output_Params[3] AND Robot.Outputs.MotionCommand.Argument3 = Output_Params[4] AND Robot.Outputs.MotionCommand.Argument4 = Output_Params[5] AND Robot.Outputs.MotionCommand.Argument5 = Output_Params[6] THEN
            IF Robot.Inputs.Motion.MoveID = Robot.Outputs.MoveID THEN
                Buffered := TRUE;
            END_IF;
        END_IF;
    END_IF;
END_IF;

(*If External _Move ID is equal to Internal, raise an error*)
IF ExternalMoveID = 32040 OR ExternalMoveID = 32041 THEN
    Error := TRUE;
END_IF;
FirstScan := TRUE;

END_FUNCTION_BLOCK

// Device/Application/F1000_FBs/Meca500/Utiliy/CalculateWRF
FUNCTION_BLOCK CalculateWRF
VAR
	Norm_uz: REAL;
	// Direction du vecteur
	Norm_ux: REAL := 1;
	ux: ARRAY[0..2] OF REAL;
	// Vecteur x selon ux
	uvx: ARRAY[0..2] OF REAL;
	// Vecteur y selon ux
	uvy: ARRAY[0..2] OF REAL;
	uz: ARRAY[0..2] OF REAL;
	Gamma_Lreal_to_REAL: REAL;
	Alpha_Lreal_to_REAL: REAL;
END_VAR
VAR_INPUT
	// Point n°1
	P1: ARRAY[0..2] OF REAL;
	// Point n°2
	P2: ARRAY[0..2] OF REAL;
	// Point n°3
	P3: ARRAY[0..2] OF REAL;
END_VAR
VAR
	//  α
	Alpha: LREAL;
	v13: ARRAY[0..2] OF REAL;
	// Angle α en degré
	Alpha_deg: REAL;
	// β
	Beta: REAL;
	// Angle β en degré
	Beta_deg: REAL;
	// γ
	Gamma: LREAL;
	// Angle γ en degré
	Gamma_deg: REAL;
END_VAR
VAR_OUTPUT
	// Coordonné WRF
	Result_WRF: ARRAY[0..5] OF REAL;
END_VAR
VAR
	Norm_v13: REAL;
	uv13: ARRAY[0..2] OF REAL;
	uvz: ARRAY[0..2] OF REAL;
END_VAR

//	Following the method available on Mecademic website : 
//	https://support.mecademic.com/en/support/solutions/articles/64000248048-how-do-i-calculate-the-wrf-using-a-3-point-method-

	  //[0]= x //[1]=y //[2]=z
       ux[0]:=(P2[0]-P1[0]); 
	   ux[1]:=(P2[1]-P1[1]); 
	   ux[2]:=(P2[2]-P1[2]); 
	
	   Norm_ux:=SQRT((ux[0]*ux[0])+(ux[1]*ux[1])+(ux[2]*ux[2]));
	   
	IF Norm_ux>10 THEN 
	   uvx[0]:=ux[0]/Norm_ux;
	   uvx[1]:=ux[1]/Norm_ux;
	   uvx[2]:=ux[2]/Norm_ux;
	END_IF
	
	   v13[0]:=(P3[0]-P1[0]);
	   v13[1]:=(P3[1]-P1[1]);
	   v13[2]:=(P3[2]-P1[2]);
	
	   Norm_v13:=SQRT((v13[0]*v13[0])+(v13[1]*v13[1])+(v13[2]*v13[2]));
	   
	IF Norm_v13> 10 THEN  
	   uv13[0]:=v13[0]/norm_v13;
	   uv13[1]:=v13[1]/norm_v13;
	   uv13[2]:=v13[2]/norm_v13;
	END_IF
	
	   uz[0]:=(uvx[1]*uv13[2])-(uvx[2]*uv13[1]); 
	   uz[1]:=(uvx[2]*uv13[0])-(uvx[0]*uv13[2]); 
	   uz[2]:=(uvx[0]*uv13[1])-(uvx[1]*uv13[0]); 
	
	IF NOT(Norm_ux<10)AND NOT(norm_v13 <10)THEN
	   Norm_uz:=SQRT((uz[0]*uz[0])+(uz[1]*uz[1])+(uz[2]*uz[2]));
	   uvz[0]:=uz[0]/norm_uz; 
	   uvz[1]:=uz[1]/norm_uz; 
	   uvz[2]:=uz[2]/norm_uz; 
	END_IF
	
	   uvy[0]:=(uvz[1]*uvx[2])-(uvz[2]*uvx[1]);
	   uvy[1]:=(uvz[2]*uvx[0])-(uvz[0]*uvx[2]); 
	   uvy[2]:=(uvz[0]*uvx[1])-(uvz[1]*uvx[0]); 
	
	IF ABS (uvz[0])=1 THEN
			Beta_deg:=uvz[0]*90;
			Gamma:= MATH.atan2(lrSinus:= uvY[0], lrCosinus:=uvX[0] );
			
		    Gamma_Lreal_to_REAL:=LREAL_TO_REAL(Gamma);
			Gamma_deg:=TES.FC_RadToDeg(i_rRad:=Gamma_Lreal_to_REAL );  
			Alpha_deg:=0;
	ELSE
			Beta:=ASIN(uvz[0]);
			Beta_deg:=TES.FC_RadToDeg(i_rRad:=Beta );
			Gamma:= MATH.atan2(lrSinus:= -uvy[0], lrCosinus:= uvx[0]);
			Gamma_Lreal_to_REAL:=LREAL_TO_REAL(Gamma);
			Gamma_deg:=TES.FC_RadToDeg(i_rRad:=Gamma_Lreal_to_REAL ); 
			Alpha:= MATH.atan2(lrSinus:=-uvz[1] , lrCosinus:=uvz[2]);
			Alpha_Lreal_to_REAL:=LREAL_TO_REAL(Alpha);
			Alpha_deg:=TES.FC_RadToDeg(i_rRad:=Alpha_Lreal_to_REAL );
	END_IF
	
			Result_WRF[0]:=P1[0];      // x    
			Result_WRF[1]:=P1[1];      // y
			Result_WRF[2]:=P1[2];      // z
			Result_WRF[3]:=alpha_deg;  // α
			Result_WRF[4]:=beta_deg;   // β
			Result_WRF[5]:=gamma_deg;  // γ

END_FUNCTION_BLOCK

// Device/Application/F001_ROBOT/F001_SR02_RBT_ERRORS
PROGRAM F001_SR02_RBT_ERRORS
VAR
END_VAR

(* body of a kind this reader does not render *)

END_PROGRAM

// Device/Application/F001_ROBOT/F001_SR03_STEPS
PROGRAM F001_SR03_STEPS
VAR
	TON1: TON;
	TON2: ton;
	TON3: ton;
	TON4: ton;
	TON5: ton;
END_VAR

(* body of a kind this reader does not render *)

END_PROGRAM

// Device/Application/F001_ROBOT/F001_SR04_RBT_INIT
PROGRAM F001_SR04_RBT_INIT
VAR
	Buffered: BOOL;
	Sent: BOOL;
	SetCartLinVel1: SetCartLinVel;
	SetJointVel1: SetJointVel;
	SETLinVEL: BOOL;
	SetJtVel: BOOL;
END_VAR

(* body of a kind this reader does not render *)

END_PROGRAM

// Device/Application/F1000_FBs/Meca500/SetJointVel
FUNCTION_BLOCK SetJointVel
VAR_INPUT
	Velocity_Percentage					:	REAL;
	ExternalStatecontrol 	:	BOOL;
	ExternalMoveID			:	UINT;
END_VAR
VAR_IN_OUT
	Robot	:	Meca500;	
	Sent		:	BOOL;
	Buffered	:	BOOL;
END_VAR
VAR_OUTPUT
	Error		:	BOOL;
END_VAR
VAR
	Output_Params	:	ARRAY[1..6] OF REAL;
	FirstScan		:	Bool;
END_VAR

        (*Collect Inputs and store them locally*)
Output_Params[1]:=Velocity_Percentage;
Output_Params[2]:=0;
Output_Params[3]:=0;
Output_Params[4]:=0;
Output_Params[5]:=0;
Output_Params[6]:=0;


(* If Values have change, Reinitialise Outputs*)

IF FirstScan=0 OR Robot.Outputs.MotionCommand.Argument0 <> Output_Params[1] OR Robot.Outputs.MotionCommand.Argument1 <> Output_Params[2] OR Robot.Outputs.MotionCommand.Argument2 <> Output_Params[3] OR Robot.Outputs.MotionCommand.Argument3 <> Output_Params[4] OR Robot.Outputs.MotionCommand.Argument4 <> Output_Params[5] OR Robot.Outputs.MotionCommand.Argument5 <> Output_Params[6] THEN
	Buffered := FALSE;
	Sent := FALSE;
END_IF;

(*if not in legacy mode, Act Setpoint*)
IF Robot.Outputs.MoveID <> 0 THEN
    Robot.Outputs.MotionControl.SetPoint := TRUE;
END_IF;

(* To send _Move, send _Move ID *)
IF NOT Buffered AND NOT Sent THEN
    
    Robot.Outputs.MotionCommand.MoveCommand := Meca500_MotionCommandID.SET_JOINT_VEL;
    Robot.Outputs.MotionCommand.Argument0 := Output_Params[1];
	Robot.Outputs.MotionCommand.Argument1 := Output_Params[2];
	Robot.Outputs.MotionCommand.Argument2 := Output_Params[3];
	Robot.Outputs.MotionCommand.Argument3 := Output_Params[4];
	Robot.Outputs.MotionCommand.Argument4 := Output_Params[5];
	Robot.Outputs.MotionCommand.Argument5 := Output_Params[6];
    
    IF ExternalStateControl THEN
        IF ExternalMoveID <> 0 AND ExternalMoveID <> 32080 AND ExternalMoveID <> 32081 THEN
            Robot.Outputs.MoveID := ExternalMoveID;
            Sent := TRUE;
        END_IF;
        
    ELSE (*Not External Control*)
        IF Robot.Outputs.MoveID = 32080 THEN
            Robot.Outputs.MoveID := 32081;
        ELSIF Robot.Outputs.MoveID = 32081 THEN
            Robot.Outputs.MoveID := 32080;
        ELSIF Robot.Outputs.MoveID <> 32080 OR Robot.Outputs.MoveID <> 32081 THEN
            Robot.Outputs.MoveID := 32080;
        END_IF;
        Sent := TRUE;
    END_IF;
END_IF;

(* Check if _Move has been sent, if so, check if it was received *)
IF Sent THEN
    IF Robot.Outputs.MotionCommand.MoveCommand = Meca500_MotionCommandID.SET_JOINT_VEL THEN
        IF Robot.Outputs.MotionCommand.Argument0 = Output_Params[1] AND Robot.Outputs.MotionCommand.Argument1 = Output_Params[2] AND Robot.Outputs.MotionCommand.Argument2 = Output_Params[3] AND Robot.Outputs.MotionCommand.Argument3 = Output_Params[4] AND Robot.Outputs.MotionCommand.Argument4 = Output_Params[5] AND Robot.Outputs.MotionCommand.Argument5 = Output_Params[6] THEN
            IF Robot.Inputs.Motion.MoveID = Robot.Outputs.MoveID THEN
                Buffered := TRUE;
            END_IF;
        END_IF;
    END_IF;
END_IF;

(*If External _Move ID is equal to Internal, raise an error*)
IF ExternalMoveID = 32080 OR ExternalMoveID = 32081 THEN
    Error := TRUE;
END_IF;
FirstScan:=TRUE;

END_FUNCTION_BLOCK

// Device/Application/F001_ROBOT/F001_SR05_SET_TRF
PROGRAM F001_SR05_SET_TRF
VAR
	
	Sent: BOOL;
	Buffered: BOOL;
	SetTrf1: SetTrf;
	Error: BOOL;
	TrfPose: ARRAY [1..6] OF REAL:=[0,0,0,0,0,0];
END_VAR

(* body of a kind this reader does not render *)

END_PROGRAM

// Device/Application/F1000_FBs/Meca500/SetTrf
FUNCTION_BLOCK SetTrf
VAR_INPUT
	Pose					:	ARRAY[1..6]OF REAL;
	ExternalStatecontrol 	:	BOOL;
	ExternalMoveID			:	UINT;
END_VAR
VAR_IN_OUT
	Robot	:	Meca500;	
	Sent		:	BOOL;
	Buffered	:	BOOL;
END_VAR
VAR_OUTPUT
	Error		:	BOOL;
END_VAR
VAR
	Output_Params	:	ARRAY[1..6] OF REAL;
	FirstScan		:	Bool;
END_VAR

        (*Collect Inputs and store them locally*)
Output_Params[1]:=Pose[1];
Output_Params[2]:=Pose[2];
Output_Params[3]:=Pose[3];
Output_Params[4]:=Pose[4];
Output_Params[5]:=Pose[5];
Output_Params[6]:=Pose[6];

(* If Values have change, Reinitialise Outputs*)

IF FirstScan=0 OR Robot.Outputs.MotionCommand.Argument0 <> Output_Params[1] OR Robot.Outputs.MotionCommand.Argument1 <> Output_Params[2] OR Robot.Outputs.MotionCommand.Argument2 <> Output_Params[3] OR Robot.Outputs.MotionCommand.Argument3 <> Output_Params[4] OR Robot.Outputs.MotionCommand.Argument4 <> Output_Params[5] OR Robot.Outputs.MotionCommand.Argument5 <> Output_Params[6] THEN
	Buffered := FALSE;
	Sent := FALSE;
END_IF;


(*if not in legacy mode, Act Setpoint*)
IF Robot.Outputs.MoveID <> 0 THEN
    Robot.Outputs.MotionControl.SetPoint := TRUE;
END_IF;

(* To send _Move, send _Move ID *)
IF NOT Buffered AND NOT Sent THEN
    
    Robot.Outputs.MotionCommand.MoveCommand := Meca500_MotionCommandID.SET_TRF;
    Robot.Outputs.MotionCommand.Argument0 := Output_Params[1];
	Robot.Outputs.MotionCommand.Argument1 := Output_Params[2];
	Robot.Outputs.MotionCommand.Argument2 := Output_Params[3];
	Robot.Outputs.MotionCommand.Argument3 := Output_Params[4];
	Robot.Outputs.MotionCommand.Argument4 := Output_Params[5];
	Robot.Outputs.MotionCommand.Argument5 := Output_Params[6];
    
    IF ExternalStateControl THEN
        IF ExternalMoveID <> 0 AND ExternalMoveID <> 32130 AND ExternalMoveID <> 32131 THEN
            Robot.Outputs.MoveID := ExternalMoveID;
            Sent := TRUE;
        END_IF;
        
    ELSE (*Not External Control*)
        IF Robot.Outputs.MoveID = 32130 THEN
            Robot.Outputs.MoveID := 32131;
        ELSIF Robot.Outputs.MoveID = 32131 THEN
            Robot.Outputs.MoveID := 32130;
        ELSIF Robot.Outputs.MoveID <> 32130 OR Robot.Outputs.MoveID <> 32131 THEN
            Robot.Outputs.MoveID := 32130;
        END_IF;
        Sent := TRUE;
    END_IF;
END_IF;

(* Check if _Move has been sent, if so, check if it was received *)
IF Sent THEN
    IF Robot.Outputs.MotionCommand.MoveCommand = Meca500_MotionCommandID.SET_TRF THEN
        IF Robot.Outputs.MotionCommand.Argument0 = Output_Params[1] AND Robot.Outputs.MotionCommand.Argument1 = Output_Params[2] AND Robot.Outputs.MotionCommand.Argument2 = Output_Params[3] AND Robot.Outputs.MotionCommand.Argument3 = Output_Params[4] AND Robot.Outputs.MotionCommand.Argument4 = Output_Params[5] AND Robot.Outputs.MotionCommand.Argument5 = Output_Params[6] THEN
            IF Robot.Inputs.Motion.MoveID = Robot.Outputs.MoveID THEN
                Buffered := TRUE;
            END_IF;
        END_IF;
    END_IF;
END_IF;

(*If External _Move ID is equal to Internal, raise an error*)
IF ExternalMoveID = 32130 OR ExternalMoveID = 32131 THEN
    Error := TRUE;
END_IF;
FirstScan:=TRUE;

END_FUNCTION_BLOCK

// Device/Application/F001_ROBOT/F001_SR06_RBT_MOTIONS
PROGRAM F001_SR06_RBT_MOTIONS
VAR
	
	HomePos:ARRAY[0..5]OF REAL := [55, -48, -15, 92.7, -43, -185];
	ApproachPos:ARRAY[0..5]OF REAL := [41.73, 23.68, -29.2, -83, 42, -8.26];
	BY_PASS: ARRAY[0..10] OF bool;
END_VAR
VAR_INPUT
	PickPos1:ARRAY[0..5]OF REAL := [0, 0, 0, 0, 0, 0];
	PickPos2:ARRAY[0..5]OF REAL := [0, 0, 0, 0, 0, 0];
END_VAR
VAR
	MovePose:ARRAY[0..5]OF Movepose;
	MoveJoints:ARRAY[0..5]OF MoveJoints;

	Buffered: BOOL;
	Sent: BOOL;
	SetCheckPoint1: ARRAY[0..5] OF SetCheckpoint;
	MoveLinRelTrf1: ARRAY[0..5] OF MoveLinRelTrf;
END_VAR

(* body of a kind this reader does not render *)

END_PROGRAM

// Device/Application/F001_ROBOT/F001_SR07_CAMERA
PROGRAM F001_SR07_CAMERA
VAR
END_VAR

(* body of a kind this reader does not render *)

END_PROGRAM

// Device/Application/F001_ROBOT/F001_SR08_Explicit
PROGRAM F001_SR08_Explicit
VAR
END_VAR

END_PROGRAM

// Device/Application/F001_ROBOT/F001_SR08_Explicit_Messaging
PROGRAM F001_SR08_Explicit_Messaging
VAR
    // State machine control
    iState       : INT := 0; 
    iIndex       : WORD := 1; // Cycles from 1 to 6
    
    // Local array buffer to hold the 6 camera values
    aWriteValues : ARRAY[1..6] OF REAL; 
    
    // Active buffer variable for the current pointer address
    rCurrentValue : REAL;
    
    // Pure ST Instance of the EtherNet/IP Function Block
    fbSetAttributeSingle : ENIP.Set_Attribute_Single;
END_VAR

CASE iState OF
    
    0: (* IDLE STATE: Wait for the user trigger *)
        IF GVL.Explicit.xTriggerWrite THEN
            // 1. Snapshot the live GVL values into our local loop array
            aWriteValues[1] := GVL.CAM_1.RESULT_POSX;
            aWriteValues[2] := GVL.CAM_1.RESULT_POSY;
            aWriteValues[3] := GVL.CAM_1.RESULT_POSZ;
            aWriteValues[4] := GVL.CAM_1.RESULT_POSRX;
            aWriteValues[5] := GVL.CAM_1.RESULT_POSRY;
            aWriteValues[6] := GVL.CAM_1.RESULT_POSRZ;
            
            // 2. Set up initial loop states
            iIndex := 1;          // Start at Attribute 1 (X)
            
            // 3. Clear global status flags before starting
            GVL.Explicit.xWriteDone  := FALSE;
            GVL.Explicit.xWriteError := FALSE;
            
            iState := 10;         // Move to transmission step
        END_IF
        
    10: (* PREPARE DATA: Load value and fire execution pulse *)
        rCurrentValue := aWriteValues[iIndex];
        
        // Lower the user trigger immediately so it doesn't loop infinitely
        GVL.Explicit.xTriggerWrite := FALSE; 
        
        // Execute the block with the current index mapped to wAttribute
        fbSetAttributeSingle(
            xExecute            := TRUE,
            itfEtherNetIPDevice := FANUC_Robot,
            eClass              := 16#6C,             // Position Register Class
            dwInstance          := 1,                 // Target PR[1] on the Fanuc
            wAttribute          := iIndex,            // Cycles 1 to 6 (X, Y, Z, RX, RY, RZ)
            tTimeOut            := T#1s,
            pData               := ADR(rCurrentValue),
            udiDataSize         := 4,                 // 4 bytes for REAL
            
            xBusy               => GVL.Explicit.xWriteBusy,
            eError              => GVL.Explicit.eWriteErrorCode
        );
        
        iState := 20; // Transition to wait state

    20: (* WAIT FOR FB HANDSHAKE *)
        // Keep processing the block cyclically
        fbSetAttributeSingle();
        
        IF fbSetAttributeSingle.xDone THEN
            // Turn off xExecute to reset the FB's internal edge detector for the next run
            fbSetAttributeSingle(xExecute := FALSE); 
            
            IF iIndex >= 6 THEN
                iState := 100; // All 6 values successfully sent to the PR
            ELSE
                iIndex := iIndex + 1; // Move to the next attribute register
                iState := 10;         // Loop back to send the next coordinate
            END_IF
            
        ELSIF fbSetAttributeSingle.xError THEN
            // Capture error state, turn off execution flag, and jump to fault handling
            fbSetAttributeSingle(xExecute := FALSE);
            iState := 999; 
        END_IF

    100: (* SEQUENCE COMPLETE *)
        GVL.Explicit.xWriteDone := TRUE; 
        iState := 0; // Return smoothly to Idle, waiting for next trigger

    999: (* FAULT HANDLING *)
        GVL.Explicit.xWriteError := TRUE;
        // Logic can stop here or you can clear and return to 0 depending on recovery needs
        // iState := 0; 
        
END_CASE

END_PROGRAM

// Device/Application/F001_ROBOT/F001_SR08_ExplicitMessaging
PROGRAM F001_SR08_ExplicitMessaging
VAR
	Explicit_Send: ENIP.Set_Attribute_Single;
END_VAR

(* body of a kind this reader does not render *)

END_PROGRAM

// Device/Application/F001_ROBOT/RobotHandshake
FUNCTION_BLOCK RobotHandshake
VAR_INPUT
    xExecute      : BOOL;    // Kicked off by the Scheduler when it's time to talk
    iCommandID    : INT;     // The Command number to send (e.g., 3)
END_VAR
VAR_OUTPUT
    xBusy         : BOOL;    // Handshake sequence is running
    xDone         : BOOL;    // Handshake completed successfully
    xError        : BOOL;    // Handshake faulted / timed out
END_VAR
VAR
    iHandshakeState : INT := 0;
    tonTimeout      : TON;   // Safety timer so the PLC doesn't hang if the robot faults
END_VAR

// Safety Timeout: If the robot gets stuck mid-handshake for more than 30 seconds, trip a fault
tonTimeout(IN := (iHandshakeState > 0 AND iHandshakeState < 100), PT := T#30s);
IF tonTimeout.Q THEN
    iHandshakeState := 999;
END_IF

CASE iHandshakeState OF

    0: (* IDLE *)
        xDone  := FALSE;
        xBusy  := FALSE;
        
        IF xExecute THEN
            xBusy := TRUE;
            xError := FALSE;
            iHandshakeState := 10;
        END_IF;

    10: (* STEP 1: Fire Explicit Message to Write Coords *)
        // Kick off your explicit messaging routine 
        GVL.Explicit.xTriggerWrite := TRUE; 
        iHandshakeState := 15;

    15: (* STEP 1.5: Wait for Explicit Write to Complete *)
        // Assumes your explicit messaging block sets xTriggerWrite back to FALSE when done.
        // If it uses a separate "Done" flag (e.g., GVL.Explicit.xWriteDone), use that here instead!
        IF NOT GVL.Explicit.xTriggerWrite THEN
            // Coords are successfully in the Fanuc registers! Now send the execution command.
            GVL.Robot.CMD := INT_TO_BYTE(iCommandID); 
            iHandshakeState := 20;
        END_IF;

    20: (* STEP 2: Wait for Robot Echo AND ensure previous Complete flag is dropped *)
        // Since we aren't using a BUSY bit, we must ensure the robot echoes our command 
        // AND its COMPLETE byte has dropped back to 0. This prevents skipping steps!
        IF (GVL.Robot.ECHO = GVL.Robot.CMD) AND (GVL.Robot.COMPLETE = 0) THEN
            iHandshakeState := 40;
        END_IF;

    40: (* STEP 4: Wait for Robot Completion *)
        // Wait until the robot sets its COMPLETE byte to 1
        IF GVL.Robot.COMPLETE = 1 THEN
            GVL.Robot.ACK_Complete := 1; // Send 1 (True) as a byte to ACK the robot
            iHandshakeState := 50;
        END_IF;

    50: (* STEP 5: Interlocking Reset *)
        // Wait for the robot to see our ACK and clear its COMPLETE byte back to 0
        IF GVL.Robot.COMPLETE = 0 THEN
            GVL.Robot.ACK_Complete := 0; // Clear our acknowledgement byte back to 0
            GVL.Robot.CMD          := 0; // Reset our command register byte back to 0
            iHandshakeState        := 100;
        END_IF;

    100: (* HANDSHAKE COMPLETE *)
        xBusy := FALSE;
        xDone := TRUE;
        
        // Wait for the master scheduler to drop xExecute before dropping back to IDLE
        IF NOT xExecute THEN
            iHandshakeState := 0;
        END_IF;

    999: (* FAULT HANDLING *)
        xBusy  := FALSE;
        xError := TRUE;
        
